LIN {X 0,Y 539.25,Z 1008.036,A -85,B 0,C 180,E1 3968.069,E2 3968.069} C_VEL
LIN {X 0,Y 539.667,Z 991.588,A -85,B 0,C 180,E1 3971.094,E2 3971.094} C_VEL
LIN {X 0,Y 540.295,Z 970.206,A -85,B 0,C 180,E1 3973.778,E2 3973.778} C_VEL
LIN {X 0,Y 541.178,Z 945.142,A -85,B 0,C 180,E1 3975.97,E2 3975.97} C_VEL
LIN {X 0,Y 542.037,Z 916.074,A -85,B 0,C 180,E1 3977.682,E2 3977.682} C_VEL
LIN {X 0,Y 542.64,Z 884.653,A -85,B 0,C 180,E1 3978.783,E2 3978.783} C_VEL
LIN {X 0,Y 541.923,Z 855.869,A -85,B 0,C 180,E1 3979.307,E2 3979.307} C_VEL
LIN {X 0,Y 538.385,Z 843.44,A -85,B 0,C 180,E1 3979.641,E2 3979.641} C_VEL
LIN {X 0,Y 538.323,Z 843.44,A -85,B 0,C 180,E1 3984.951,E2 3984.951} C_VEL
LIN {X 0,Y 538.286,Z 843.44,A -85,B 0,C 180,E1 3990.414,E2 3990.414} C_VEL
LIN {X 0,Y 538.342,Z 843.44,A -85,B 0,C 180,E1 3996.196,E2 3996.196} C_VEL
LIN {X 0,Y 538.103,Z 843.44,A -85,B 0,C 180,E1 4002.471,E2 4002.471} C_VEL
LIN {X 0,Y 538.121,Z 843.44,A -85,B 0,C 180,E1 4007.522,E2 4007.522} C_VEL
LIN {X 0,Y 538.444,Z 843.44,A -85,B 0,C 180,E1 4013.804,E2 4013.804} C_VEL
LIN {X 0,Y 538.555,Z 844.13,A -85,B 0,C 180,E1 4016.198,E2 4016.198} C_VEL
LIN {X 0,Y 549.167,Z 867.562,A -85,B 0,C 180,E1 4017.292,E2 4017.292} C_VEL
LIN {X 0,Y 548.845,Z 915.281,A -85,B 0,C 180,E1 4018.203,E2 4018.203} C_VEL
LIN {X 0,Y 547.509,Z 954.361,A -85,B 0,C 180,E1 4019.575,E2 4019.575} C_VEL
LIN {X 0,Y 545.893,Z 988.921,A -85,B 0,C 180,E1 4021.38,E2 4021.38} C_VEL
LIN {X 0,Y 543.954,Z 1023.542,A -85,B 0,C 180,E1 4023.86,E2 4023.86} C_VEL
LIN {X 0,Y 542.252,Z 1054.192,A -85,B 0,C 180,E1 4026.77,E2 4026.77} C_VEL
LIN {X 0,Y 540.773,Z 1081.673,A -85,B 0,C 180,E1 4030.169,E2 4030.169} C_VEL
LIN {X 0,Y 539.773,Z 1104.705,A -85,B 0,C 180,E1 4033.918,E2 4033.918} C_VEL
LIN {X 0,Y 539.188,Z 1122.492,A -85,B 0,C 180,E1 4037.841,E2 4037.841} C_VEL
LIN {X 0,Y 539.047,Z 1134.255,A -85,B 0,C 180,E1 4041.519,E2 4041.519} C_VEL
LIN {X 0,Y 538.908,Z 1141.5,A -85,B 0,C 180,E1 4045.164,E2 4045.164} C_VEL
LIN {X 0,Y 538.866,Z 1144.612,A -85,B 0,C 180,E1 4048.389,E2 4048.389} C_VEL
LIN {X 0,Y 538.972,Z 1144.555,A -85,B 0,C 180,E1 4051.609,E2 4051.609} C_VEL
LIN {X 0,Y 538.984,Z 1140.149,A -85,B 0,C 180,E1 4055.642,E2 4055.642} C_VEL
LIN {X 0,Y 539.118,Z 1130.585,A -85,B 0,C 180,E1 4059.701,E2 4059.701} C_VEL
LIN {X 0,Y 539.5,Z 1115.458,A -85,B 0,C 180,E1 4063.786,E2 4063.786} C_VEL
LIN {X 0,Y 540.206,Z 1095.274,A -85,B 0,C 180,E1 4067.665,E2 4067.665} C_VEL
LIN {X 0,Y 541.512,Z 1068.316,A -85,B 0,C 180,E1 4071.506,E2 4071.506} C_VEL
LIN {X 0,Y 543.119,Z 1038.564,A -85,B 0,C 180,E1 4074.719,E2 4074.719} C_VEL
LIN {X 0,Y 545.035,Z 1004.579,A -85,B 0,C 180,E1 4077.497,E2 4077.497} C_VEL
LIN {X 0,Y 546.848,Z 969.441,A -85,B 0,C 180,E1 4079.619,E2 4079.619} C_VEL
LIN {X 0,Y 548.311,Z 933.853,A -85,B 0,C 180,E1 4081.138,E2 4081.138} C_VEL
LIN {X 0,Y 549.352,Z 895.087,A -85,B 0,C 180,E1 4082.16,E2 4082.16} C_VEL
LIN {X 0,Y 548.858,Z 867.054,A -85,B 0,C 180,E1 4082.647,E2 4082.647} C_VEL
LIN {X 0,Y 538.256,Z 843.44,A -85,B 0,C 180,E1 4083.79,E2 4083.79} C_VEL
LIN {X 0,Y 538.332,Z 843.44,A -85,B 0,C 180,E1 4088.226,E2 4088.226} C_VEL
LIN {X 0,Y 538.212,Z 843.44,A -85,B 0,C 180,E1 4094.693,E2 4094.693} C_VEL
LIN {X 0,Y 538.217,Z 843.44,A -85,B 0,C 180,E1 4099.688,E2 4099.688} C_VEL
LIN {X 0,Y 538.184,Z 843.44,A -85,B 0,C 180,E1 4105.764,E2 4105.764} C_VEL
LIN {X 0,Y 538.293,Z 843.44,A -85,B 0,C 180,E1 4111.438,E2 4111.438} C_VEL
LIN {X 0,Y 538.435,Z 843.44,A -85,B 0,C 180,E1 4116.819,E2 4116.819} C_VEL
LIN {X 0,Y 538.559,Z 843.44,A -85,B 0,C 180,E1 4121.989,E2 4121.989} C_VEL
LIN {X 0,Y 538.664,Z 843.44,A -85,B 0,C 180,E1 4127.007,E2 4127.007} C_VEL
LIN {X 0,Y 538.668,Z 843.44,A -85,B 0,C 180,E1 4131.922,E2 4131.922} C_VEL
LIN {X 0,Y 538.803,Z 843.44,A -85,B 0,C 180,E1 4136.779,E2 4136.779} C_VEL
LIN {X 0,Y 538.914,Z 843.44,A -85,B 0,C 180,E1 4141.611,E2 4141.611} C_VEL
LIN {X 0,Y 538.794,Z 843.44,A -85,B 0,C 180,E1 4146.454,E2 4146.454} C_VEL
LIN {X 0,Y 538.518,Z 843.44,A -85,B 0,C 180,E1 4152.998,E2 4152.998} C_VEL
LIN {X 0,Y 538.458,Z 843.44,A -85,B 0,C 180,E1 4158.017,E2 4158.017} C_VEL
LIN {X 0,Y 538.431,Z 843.44,A -85,B 0,C 180,E1 4163.182,E2 4163.182} C_VEL
LIN {X 0,Y 538.42,Z 843.44,A -85,B 0,C 180,E1 4165.122,E2 4165.122} C_VEL
LIN {X 0,Y 537.116,Z 843.44,A -85,B 0,C 180,E1 4166.044,E2 4166.044} C_VEL
LIN {X 0,Y 530.442,Z 843.44,A -85,B 0,C 180,E1 4168.554,E2 4168.554} C_VEL
LIN {X 0,Y 530.36,Z 843.44,A -85,B 0,C 180,E1 4168.792,E2 4168.792} C_VEL
LIN {X 0,Y 530.3,Z 843.44,A -85,B 0,C 180,E1 4174.819,E2 4174.819} C_VEL
LIN {X 0,Y 530.294,Z 843.44,A -85,B 0,C 180,E1 4181.044,E2 4181.044} C_VEL
LIN {X 0,Y 530.296,Z 843.44,A -85,B 0,C 180,E1 4186.745,E2 4186.745} C_VEL
LIN {X 0,Y 530.38,Z 844.061,A -85,B 0,C 180,E1 4190.548,E2 4190.548} C_VEL
LIN {X 0,Y 546.247,Z 875.945,A -85,B 0,C 180,E1 4192.425,E2 4192.425} C_VEL
LIN {X 0,Y 545.089,Z 919.849,A -85,B 0,C 180,E1 4193.364,E2 4193.364} C_VEL
LIN {X 0,Y 543.337,Z 959.293,A -85,B 0,C 180,E1 4194.829,E2 4194.829} C_VEL
LIN {X 0,Y 541.124,Z 997.278,A -85,B 0,C 180,E1 4196.867,E2 4196.867} C_VEL
LIN {X 0,Y 538.391,Z 1035.857,A -85,B 0,C 180,E1 4199.684,E2 4199.684} C_VEL
LIN {X 0,Y 535.813,Z 1071.337,A -85,B 0,C 180,E1 4203.12,E2 4203.12} C_VEL
LIN {X 0,Y 533.767,Z 1102.204,A -85,B 0,C 180,E1 4207.015,E2 4207.015} C_VEL
LIN {X 0,Y 532.286,Z 1127.302,A -85,B 0,C 180,E1 4211.122,E2 4211.122} C_VEL
LIN {X 0,Y 531.574,Z 1145.987,A -85,B 0,C 180,E1 4215.147,E2 4215.147} C_VEL
LIN {X 0,Y 531.16,Z 1160,A -85,B 0,C 180,E1 4219.272,E2 4219.272} C_VEL
LIN {X 0,Y 531.066,Z 1169.479,A -85,B 0,C 180,E1 4223.452,E2 4223.452} C_VEL
LIN {X 0,Y 530.978,Z 1173.628,A -85,B 0,C 180,E1 4226.731,E2 4226.731} C_VEL
LIN {X 0,Y 530.953,Z 1175,A -85,B 0,C 180,E1 4230.001,E2 4230.001} C_VEL
LIN {X 0,Y 530.956,Z 1173.247,A -85,B 0,C 180,E1 4233.638,E2 4233.638} C_VEL
LIN {X 0,Y 531.102,Z 1166.328,A -85,B 0,C 180,E1 4238.196,E2 4238.196} C_VEL
LIN {X 0,Y 531.263,Z 1155.088,A -85,B 0,C 180,E1 4242.343,E2 4242.343} C_VEL
LIN {X 0,Y 531.834,Z 1138.762,A -85,B 0,C 180,E1 4246.542,E2 4246.542} C_VEL
LIN {X 0,Y 532.945,Z 1116.87,A -85,B 0,C 180,E1 4250.718,E2 4250.718} C_VEL
LIN {X 0,Y 534.62,Z 1089.193,A -85,B 0,C 180,E1 4254.753,E2 4254.753} C_VEL
LIN {X 0,Y 536.83,Z 1057.678,A -85,B 0,C 180,E1 4258.313,E2 4258.313} C_VEL
LIN {X 0,Y 539.421,Z 1021.619,A -85,B 0,C 180,E1 4261.454,E2 4261.454} C_VEL
LIN {X 0,Y 542.046,Z 982.156,A -85,B 0,C 180,E1 4264.028,E2 4264.028} C_VEL
LIN {X 0,Y 544.325,Z 941.057,A -85,B 0,C 180,E1 4265.927,E2 4265.927} C_VEL
LIN {X 0,Y 545.815,Z 903.152,A -85,B 0,C 180,E1 4267.057,E2 4267.057} C_VEL
LIN {X 0,Y 545.931,Z 873.898,A -85,B 0,C 180,E1 4267.634,E2 4267.634} C_VEL
LIN {X 0,Y 530.636,Z 845.115,A -85,B 0,C 180,E1 4269.411,E2 4269.411} C_VEL
LIN {X 0,Y 530.457,Z 843.44,A -85,B 0,C 180,E1 4269.456,E2 4269.456} C_VEL
LIN {X 0,Y 530.126,Z 843.44,A -85,B 0,C 180,E1 4275.566,E2 4275.566} C_VEL
LIN {X 0,Y 530.325,Z 843.44,A -85,B 0,C 180,E1 4281.093,E2 4281.093} C_VEL
LIN {X 0,Y 530.43,Z 843.44,A -85,B 0,C 180,E1 4287.159,E2 4287.159} C_VEL
LIN {X 0,Y 530.426,Z 843.44,A -85,B 0,C 180,E1 4292.827,E2 4292.827} C_VEL
LIN {X 0,Y 530.381,Z 843.44,A -85,B 0,C 180,E1 4298.217,E2 4298.217} C_VEL
LIN {X 0,Y 530.241,Z 843.44,A -85,B 0,C 180,E1 4299.962,E2 4299.962} C_VEL
LIN {X 0,Y 535.362,Z 865.662,A -85,B 0,C 180,E1 4300.493,E2 4300.493} C_VEL
LIN {X 0,Y 534.887,Z 898.665,A -85,B 0,C 180,E1 4301.266,E2 4301.266} C_VEL
LIN {X 0,Y 534.068,Z 927.663,A -85,B 0,C 180,E1 4302.577,E2 4302.577} C_VEL
LIN {X 0,Y 533.058,Z 956.085,A -85,B 0,C 180,E1 4304.579,E2 4304.579} C_VEL
LIN {X 0,Y 532.241,Z 978.331,A -85,B 0,C 180,E1 4306.846,E2 4306.846} C_VEL
LIN {X 0,Y 531.653,Z 997.827,A -85,B 0,C 180,E1 4309.667,E2 4309.667} C_VEL
LIN {X 0,Y 531.371,Z 1011.704,A -85,B 0,C 180,E1 4312.633,E2 4312.633} C_VEL
LIN {X 0,Y 531.191,Z 1020.396,A -85,B 0,C 180,E1 4315.596,E2 4315.596} C_VEL
LIN {X 0,Y 531.1,Z 1024.385,A -85,B 0,C 180,E1 4318.366,E2 4318.366} C_VEL
LIN {X 0,Y 531.096,Z 1024.309,A -85,B 0,C 180,E1 4321.633,E2 4321.633} C_VEL
LIN {X 0,Y 531.2,Z 1019.034,A -85,B 0,C 180,E1 4324.904,E2 4324.904} C_VEL
LIN {X 0,Y 531.382,Z 1008.039,A -85,B 0,C 180,E1 4328.189,E2 4328.189} C_VEL
LIN {X 0,Y 531.844,Z 991.591,A -85,B 0,C 180,E1 4331.26,E2 4331.26} C_VEL
LIN {X 0,Y 532.563,Z 970.21,A -85,B 0,C 180,E1 4333.982,E2 4333.982} C_VEL
LIN {X 0,Y 533.528,Z 944.229,A -85,B 0,C 180,E1 4336.272,E2 4336.272} C_VEL
LIN {X 0,Y 534.512,Z 914.964,A -85,B 0,C 180,E1 4337.993,E2 4337.993} C_VEL
LIN {X 0,Y 535.152,Z 885.089,A -85,B 0,C 180,E1 4339.045,E2 4339.045} C_VEL
LIN {X 0,Y 534.775,Z 858.414,A -85,B 0,C 180,E1 4339.54,E2 4339.54} C_VEL
LIN {X 0,Y 530.44,Z 843.44,A -85,B 0,C 180,E1 4339.92,E2 4339.92} C_VEL
LIN {X 0,Y 530.42,Z 843.44,A -85,B 0,C 180,E1 4345.348,E2 4345.348} C_VEL
LIN {X 0,Y 530.335,Z 843.44,A -85,B 0,C 180,E1 4351.071,E2 4351.071} C_VEL
LIN {X 0,Y 530.359,Z 843.44,A -85,B 0,C 180,E1 4356.928,E2 4356.928} C_VEL
LIN {X 0,Y 530.126,Z 843.44,A -85,B 0,C 180,E1 4363.266,E2 4363.266} C_VEL
LIN {X 0,Y 530.268,Z 843.44,A -85,B 0,C 180,E1 4368.947,E2 4368.947} C_VEL
LIN {X 0,Y 530.543,Z 843.44,A -85,B 0,C 180,E1 4375.427,E2 4375.427} C_VEL
LIN {X 0,Y 530.554,Z 843.44,A -85,B 0,C 180,E1 4375.604,E2 4375.604} C_VEL
LIN {X 0,Y 542.545,Z 871.557,A -85,B 0,C 180,E1 4376.904,E2 4376.904} C_VEL
LIN {X 0,Y 542.059,Z 916.69,A -85,B 0,C 180,E1 4377.801,E2 4377.801} C_VEL
LIN {X 0,Y 540.643,Z 954.411,A -85,B 0,C 180,E1 4379.15,E2 4379.15} C_VEL
LIN {X 0,Y 538.857,Z 988.917,A -85,B 0,C 180,E1 4380.972,E2 4380.972} C_VEL
LIN {X 0,Y 536.689,Z 1023.761,A -85,B 0,C 180,E1 4383.499,E2 4383.499} C_VEL
LIN {X 0,Y 534.806,Z 1054.184,A -85,B 0,C 180,E1 4386.427,E2 4386.427} C_VEL
LIN {X 0,Y 533.143,Z 1081.644,A -85,B 0,C 180,E1 4389.869,E2 4389.869} C_VEL
LIN {X 0,Y 532.025,Z 1104.702,A -85,B 0,C 180,E1 4393.677,E2 4393.677} C_VEL
LIN {X 0,Y 531.351,Z 1122.49,A -85,B 0,C 180,E1 4397.659,E2 4397.659} C_VEL
LIN {X 0,Y 531.161,Z 1134.254,A -85,B 0,C 180,E1 4401.392,E2 4401.392} C_VEL
LIN {X 0,Y 531.02,Z 1141.499,A -85,B 0,C 180,E1 4405.092,E2 4405.092} C_VEL
LIN {X 0,Y 530.964,Z 1144.612,A -85,B 0,C 180,E1 4408.365,E2 4408.365} C_VEL
LIN {X 0,Y 531.067,Z 1144.555,A -85,B 0,C 180,E1 4411.633,E2 4411.633} C_VEL
LIN {X 0,Y 531.079,Z 1140.151,A -85,B 0,C 180,E1 4415.726,E2 4415.726} C_VEL
LIN {X 0,Y 531.244,Z 1130.587,A -85,B 0,C 180,E1 4419.846,E2 4419.846} C_VEL
LIN {X 0,Y 531.659,Z 1114.651,A -85,B 0,C 180,E1 4424.182,E2 4424.182} C_VEL
LIN {X 0,Y 532.574,Z 1093.495,A -85,B 0,C 180,E1 4428.223,E2 4428.223} C_VEL
LIN {X 0,Y 533.995,Z 1067.089,A -85,B 0,C 180,E1 4431.978,E2 4431.978} C_VEL
LIN {X 0,Y 535.838,Z 1036.864,A -85,B 0,C 180,E1 4435.244,E2 4435.244} C_VEL
LIN {X 0,Y 537.938,Z 1003.455,A -85,B 0,C 180,E1 4437.976,E2 4437.976} C_VEL
LIN {X 0,Y 539.961,Z 967.997,A -85,B 0,C 180,E1 4440.115,E2 4440.115} C_VEL
LIN {X 0,Y 541.596,Z 932.081,A -85,B 0,C 180,E1 4441.632,E2 4441.632} C_VEL
LIN {X 0,Y 542.685,Z 895.255,A -85,B 0,C 180,E1 4442.601,E2 4442.601} C_VEL
LIN {X 0,Y 542.233,Z 869.608,A -85,B 0,C 180,E1 4443.058,E2 4443.058} C_VEL
LIN {X 0,Y 530.33,Z 843.44,A -85,B 0,C 180,E1 4444.378,E2 4444.378} C_VEL
LIN {X 0,Y 530.31,Z 843.44,A -85,B 0,C 180,E1 4449.575,E2 4449.575} C_VEL
LIN {X 0,Y 530.304,Z 843.44,A -85,B 0,C 180,E1 4455.544,E2 4455.544} C_VEL
LIN {X 0,Y 530.257,Z 843.44,A -85,B 0,C 180,E1 4461.089,E2 4461.089} C_VEL
LIN {X 0,Y 530.268,Z 843.44,A -85,B 0,C 180,E1 4467.15,E2 4467.15} C_VEL
LIN {X 0,Y 530.43,Z 843.44,A -85,B 0,C 180,E1 4472.829,E2 4472.829} C_VEL
LIN {X 0,Y 530.578,Z 843.44,A -85,B 0,C 180,E1 4478.227,E2 4478.227} C_VEL
LIN {X 0,Y 530.67,Z 843.44,A -85,B 0,C 180,E1 4483.425,E2 4483.425} C_VEL
LIN {X 0,Y 530.676,Z 843.44,A -85,B 0,C 180,E1 4488.481,E2 4488.481} C_VEL
LIN {X 0,Y 530.714,Z 843.44,A -85,B 0,C 180,E1 4493.449,E2 4493.449} C_VEL
LIN {X 0,Y 530.763,Z 843.44,A -85,B 0,C 180,E1 4498.366,E2 4498.366} C_VEL
LIN {X 0,Y 530.765,Z 843.44,A -85,B 0,C 180,E1 4503.271,E2 4503.271} C_VEL
LIN {X 0,Y 530.657,Z 843.44,A -85,B 0,C 180,E1 4508.202,E2 4508.202} C_VEL
LIN {X 0,Y 530.555,Z 843.44,A -85,B 0,C 180,E1 4513.999,E2 4513.999} C_VEL
LIN {X 0,Y 530.537,Z 843.44,A -85,B 0,C 180,E1 4520.026,E2 4520.026} C_VEL
LIN {X 0,Y 530.536,Z 843.44,A -85,B 0,C 180,E1 4525.344,E2 4525.344} C_VEL
LIN {X 0,Y 530.36,Z 843.44,A -85,B 0,C 180,E1 4528.792,E2 4528.792} C_VEL
LIN {X 0,Y 527.819,Z 843.44,A -85,B 0,C 180,E1 4530.18,E2 4530.18} C_VEL
LIN {X 0,Y 522.427,Z 843.44,A -85,B 0,C 180,E1 4532.26,E2 4532.26} C_VEL
LIN {X 0,Y 522.35,Z 843.44,A -85,B 0,C 180,E1 4532.501,E2 4532.501} C_VEL
LIN {X 0,Y 522.357,Z 843.44,A -85,B 0,C 180,E1 4538.499,E2 4538.499} C_VEL
LIN {X 0,Y 522.418,Z 843.44,A -85,B 0,C 180,E1 4544.069,E2 4544.069} C_VEL
LIN {X 0,Y 522.382,Z 844.116,A -85,B 0,C 180,E1 4549.825,E2 4549.825} C_VEL
LIN {X 0,Y 539.951,Z 879.393,A -85,B 0,C 180,E1 4551.966,E2 4551.966} C_VEL
LIN {X 0,Y 538.635,Z 922.756,A -85,B 0,C 180,E1 4552.945,E2 4552.945} C_VEL
LIN {X 0,Y 536.659,Z 962.005,A -85,B 0,C 180,E1 4554.464,E2 4554.464} C_VEL
LIN {X 0,Y 534.198,Z 999.236,A -85,B 0,C 180,E1 4556.521,E2 4556.521} C_VEL
LIN {X 0,Y 531.304,Z 1036.601,A -85,B 0,C 180,E1 4559.306,E2 4559.306} C_VEL
LIN {X 0,Y 528.494,Z 1071.337,A -85,B 0,C 180,E1 4562.717,E2 4562.717} C_VEL
LIN {X 0,Y 526.312,Z 1101.078,A -85,B 0,C 180,E1 4566.498,E2 4566.498} C_VEL
LIN {X 0,Y 524.669,Z 1126.193,A -85,B 0,C 180,E1 4570.618,E2 4570.618} C_VEL
LIN {X 0,Y 523.746,Z 1145.985,A -85,B 0,C 180,E1 4574.92,E2 4574.92} C_VEL
LIN {X 0,Y 523.289,Z 1159.852,A -85,B 0,C 180,E1 4579.055,E2 4579.055} C_VEL
LIN {X 0,Y 523.163,Z 1169.479,A -85,B 0,C 180,E1 4583.353,E2 4583.353} C_VEL
LIN {X 0,Y 523.098,Z 1173.628,A -85,B 0,C 180,E1 4586.682,E2 4586.682} C_VEL
LIN {X 0,Y 523.065,Z 1175,A -85,B 0,C 180,E1 4590.001,E2 4590.001} C_VEL
LIN {X 0,Y 523.097,Z 1173.627,A -85,B 0,C 180,E1 4593.32,E2 4593.32} C_VEL
LIN {X 0,Y 523.255,Z 1167.915,A -85,B 0,C 180,E1 4597.483,E2 4597.483} C_VEL
LIN {X 0,Y 523.353,Z 1157.769,A -85,B 0,C 180,E1 4601.685,E2 4601.685} C_VEL
LIN {X 0,Y 523.901,Z 1142.484,A -85,B 0,C 180,E1 4605.937,E2 4605.937} C_VEL
LIN {X 0,Y 524.966,Z 1121.368,A -85,B 0,C 180,E1 4610.25,E2 4610.25} C_VEL
LIN {X 0,Y 526.718,Z 1095.264,A -85,B 0,C 180,E1 4614.311,E2 4614.311} C_VEL
LIN {X 0,Y 529.005,Z 1065.179,A -85,B 0,C 180,E1 4617.949,E2 4617.949} C_VEL
LIN {X 0,Y 531.717,Z 1031.06,A -85,B 0,C 180,E1 4621.158,E2 4621.158} C_VEL
LIN {X 0,Y 534.514,Z 993.918,A -85,B 0,C 180,E1 4623.82,E2 4623.82} C_VEL
LIN {X 0,Y 537.167,Z 954.369,A -85,B 0,C 180,E1 4625.886,E2 4625.886} C_VEL
LIN {X 0,Y 539.088,Z 913.257,A -85,B 0,C 180,E1 4627.323,E2 4627.323} C_VEL
LIN {X 0,Y 539.566,Z 876.644,A -85,B 0,C 180,E1 4628.111,E2 4628.111} C_VEL
LIN {X 0,Y 522.625,Z 844.942,A -85,B 0,C 180,E1 4630.139,E2 4630.139} C_VEL
LIN {X 0,Y 522.433,Z 843.44,A -85,B 0,C 180,E1 4630.286,E2 4630.286} C_VEL
LIN {X 0,Y 522.248,Z 843.44,A -85,B 0,C 180,E1 4636.455,E2 4636.455} C_VEL
LIN {X 0,Y 522.424,Z 843.44,A -85,B 0,C 180,E1 4642.513,E2 4642.513} C_VEL
LIN {X 0,Y 522.484,Z 843.44,A -85,B 0,C 180,E1 4648.562,E2 4648.562} C_VEL
LIN {X 0,Y 522.48,Z 843.44,A -85,B 0,C 180,E1 4654.237,E2 4654.237} C_VEL
LIN {X 0,Y 522.342,Z 843.44,A -85,B 0,C 180,E1 4659.689,E2 4659.689} C_VEL
LIN {X 0,Y 527.927,Z 865.615,A -85,B 0,C 180,E1 4660.207,E2 4660.207} C_VEL
LIN {X 0,Y 527.386,Z 898.235,A -85,B 0,C 180,E1 4660.976,E2 4660.976} C_VEL
LIN {X 0,Y 526.488,Z 927.634,A -85,B 0,C 180,E1 4662.317,E2 4662.317} C_VEL
LIN {X 0,Y 525.393,Z 955.804,A -85,B 0,C 180,E1 4664.326,E2 4664.326} C_VEL
LIN {X 0,Y 524.471,Z 978.32,A -85,B 0,C 180,E1 4666.647,E2 4666.647} C_VEL
LIN {X 0,Y 523.838,Z 997.943,A -85,B 0,C 180,E1 4669.532,E2 4669.532} C_VEL
LIN {X 0,Y 523.494,Z 1011.693,A -85,B 0,C 180,E1 4672.522,E2 4672.522} C_VEL
LIN {X 0,Y 523.3,Z 1020.394,A -85,B 0,C 180,E1 4675.53,E2 4675.53} C_VEL
LIN {X 0,Y 523.215,Z 1024.383,A -85,B 0,C 180,E1 4678.341,E2 4678.341} C_VEL
LIN {X 0,Y 523.212,Z 1024.308,A -85,B 0,C 180,E1 4681.657,E2 4681.657} C_VEL
LIN {X 0,Y 523.303,Z 1019.036,A -85,B 0,C 180,E1 4684.978,E2 4684.978} C_VEL
LIN {X 0,Y 523.52,Z 1008.042,A -85,B 0,C 180,E1 4688.313,E2 4688.313} C_VEL
LIN {X 0,Y 524.013,Z 992.184,A -85,B 0,C 180,E1 4691.339,E2 4691.339} C_VEL
LIN {X 0,Y 524.771,Z 972.163,A -85,B 0,C 180,E1 4693.98,E2 4693.98} C_VEL
LIN {X 0,Y 525.8,Z 947.035,A -85,B 0,C 180,E1 4696.303,E2 4696.303} C_VEL
LIN {X 0,Y 526.87,Z 918.222,A -85,B 0,C 180,E1 4698.1,E2 4698.1} C_VEL
LIN {X 0,Y 527.659,Z 888.347,A -85,B 0,C 180,E1 4699.245,E2 4699.245} C_VEL
LIN {X 0,Y 527.209,Z 859.544,A -85,B 0,C 180,E1 4699.817,E2 4699.817} C_VEL
LIN {X 0,Y 522.524,Z 843.44,A -85,B 0,C 180,E1 4700.262,E2 4700.262} C_VEL
LIN {X 0,Y 522.424,Z 843.44,A -85,B 0,C 180,E1 4706.041,E2 4706.041} C_VEL
LIN {X 0,Y 522.414,Z 843.44,A -85,B 0,C 180,E1 4711.441,E2 4711.441} C_VEL
LIN {X 0,Y 522.393,Z 843.44,A -85,B 0,C 180,E1 4717.487,E2 4717.487} C_VEL
LIN {X 0,Y 522.219,Z 843.44,A -85,B 0,C 180,E1 4723.542,E2 4723.542} C_VEL
LIN {X 0,Y 522.372,Z 843.44,A -85,B 0,C 180,E1 4728.896,E2 4728.896} C_VEL
LIN {X 0,Y 522.596,Z 843.44,A -85,B 0,C 180,E1 4734.992,E2 4734.992} C_VEL
LIN {X 0,Y 535.918,Z 873.698,A -85,B 0,C 180,E1 4736.476,E2 4736.476} C_VEL
LIN {X 0,Y 535.322,Z 917.865,A -85,B 0,C 180,E1 4737.382,E2 4737.382} C_VEL
LIN {X 0,Y 533.685,Z 956.285,A -85,B 0,C 180,E1 4738.795,E2 4738.795} C_VEL
LIN {X 0,Y 531.594,Z 992.09,A -85,B 0,C 180,E1 4740.755,E2 4740.755} C_VEL
LIN {X 0,Y 529.23,Z 1026.349,A -85,B 0,C 180,E1 4743.331,E2 4743.331} C_VEL
LIN {X 0,Y 527.099,Z 1057.721,A -85,B 0,C 180,E1 4746.475,E2 4746.475} C_VEL
LIN {X 0,Y 525.336,Z 1084.483,A -85,B 0,C 180,E1 4749.984,E2 4749.984} C_VEL
LIN {X 0,Y 524.121,Z 1106.876,A -85,B 0,C 180,E1 4753.855,E2 4753.855} C_VEL
LIN {X 0,Y 523.455,Z 1124.026,A -85,B 0,C 180,E1 4757.894,E2 4757.894} C_VEL
LIN {X 0,Y 523.244,Z 1135.215,A -85,B 0,C 180,E1 4761.68,E2 4761.68} C_VEL
LIN {X 0,Y 523.12,Z 1141.499,A -85,B 0,C 180,E1 4765.018,E2 4765.018} C_VEL
LIN {X 0,Y 523.06,Z 1144.611,A -85,B 0,C 180,E1 4768.34,E2 4768.34} C_VEL
LIN {X 0,Y 523.178,Z 1144.556,A -85,B 0,C 180,E1 4771.658,E2 4771.658} C_VEL
LIN {X 0,Y 523.189,Z 1140.152,A -85,B 0,C 180,E1 4775.813,E2 4775.813} C_VEL
LIN {X 0,Y 523.361,Z 1130.589,A -85,B 0,C 180,E1 4779.996,E2 4779.996} C_VEL
LIN {X 0,Y 523.817,Z 1115.133,A -85,B 0,C 180,E1 4784.288,E2 4784.288} C_VEL
LIN {X 0,Y 524.904,Z 1093.498,A -85,B 0,C 180,E1 4788.499,E2 4788.499} C_VEL
LIN {X 0,Y 526.412,Z 1067.473,A -85,B 0,C 180,E1 4792.264,E2 4792.264} C_VEL
LIN {X 0,Y 528.489,Z 1037.362,A -85,B 0,C 180,E1 4795.572,E2 4795.572} C_VEL
LIN {X 0,Y 530.772,Z 1004.033,A -85,B 0,C 180,E1 4798.344,E2 4798.344} C_VEL
LIN {X 0,Y 533.009,Z 968.113,A -85,B 0,C 180,E1 4800.543,E2 4800.543} C_VEL
LIN {X 0,Y 534.859,Z 931.791,A -85,B 0,C 180,E1 4802.089,E2 4802.089} C_VEL
LIN {X 0,Y 536.022,Z 894.735,A -85,B 0,C 180,E1 4803.068,E2 4803.068} C_VEL
LIN {X 0,Y 535.537,Z 872.12,A -85,B 0,C 180,E1 4803.486,E2 4803.486} C_VEL
LIN {X 0,Y 522.398,Z 843.44,A -85,B 0,C 180,E1 4805.018,E2 4805.018} C_VEL
LIN {X 0,Y 522.397,Z 843.44,A -85,B 0,C 180,E1 4811.107,E2 4811.107} C_VEL
LIN {X 0,Y 522.433,Z 843.44,A -85,B 0,C 180,E1 4816.431,E2 4816.431} C_VEL
LIN {X 0,Y 522.312,Z 843.44,A -85,B 0,C 180,E1 4822.506,E2 4822.506} C_VEL
LIN {X 0,Y 522.358,Z 843.44,A -85,B 0,C 180,E1 4828.555,E2 4828.555} C_VEL
LIN {X 0,Y 522.561,Z 843.44,A -85,B 0,C 180,E1 4834.243,E2 4834.243} C_VEL
LIN {X 0,Y 522.689,Z 843.44,A -85,B 0,C 180,E1 4839.662,E2 4839.662} C_VEL
LIN {X 0,Y 522.798,Z 843.44,A -85,B 0,C 180,E1 4844.894,E2 4844.894} C_VEL
LIN {X 0,Y 522.809,Z 843.44,A -85,B 0,C 180,E1 4851.219,E2 4851.219} C_VEL
LIN {X 0,Y 523.027,Z 843.44,A -85,B 0,C 180,E1 4856.682,E2 4856.682} C_VEL
LIN {X 0,Y 523.095,Z 843.44,A -85,B 0,C 180,E1 4861.659,E2 4861.659} C_VEL
LIN {X 0,Y 522.953,Z 843.44,A -85,B 0,C 180,E1 4866.651,E2 4866.651} C_VEL
LIN {X 0,Y 522.759,Z 843.44,A -85,B 0,C 180,E1 4871.697,E2 4871.697} C_VEL
LIN {X 0,Y 522.618,Z 843.44,A -85,B 0,C 180,E1 4877.047,E2 4877.047} C_VEL
LIN {X 0,Y 522.615,Z 843.44,A -85,B 0,C 180,E1 4882.124,E2 4882.124} C_VEL
LIN {X 0,Y 522.499,Z 843.44,A -85,B 0,C 180,E1 4887.621,E2 4887.621} C_VEL
LIN {X 0,Y 522.35,Z 843.44,A -85,B 0,C 180,E1 4892.501,E2 4892.501} C_VEL
LIN {X 0,Y 519.889,Z 843.44,A -85,B 0,C 180,E1 4893.915,E2 4893.915} C_VEL
LIN {X 0,Y 514.52,Z 843.44,A -85,B 0,C 180,E1 4896.034,E2 4896.034} C_VEL
LIN {X 0,Y 514.418,Z 843.44,A -85,B 0,C 180,E1 4896.279,E2 4896.279} C_VEL
LIN {X 0,Y 514.476,Z 843.44,A -85,B 0,C 180,E1 4902.629,E2 4902.629} C_VEL
LIN {X 0,Y 514.457,Z 843.978,A -85,B 0,C 180,E1 4909.177,E2 4909.177} C_VEL
LIN {X 0,Y 527.261,Z 868.244,A -85,B 0,C 180,E1 4910.687,E2 4910.687} C_VEL
LIN {X 0,Y 533.59,Z 880.607,A -85,B 0,C 180,E1 4911.45,E2 4911.45} C_VEL
LIN {X 0,Y 532.173,Z 925.769,A -85,B 0,C 180,E1 4912.518,E2 4912.518} C_VEL
LIN {X 0,Y 529.638,Z 969.015,A -85,B 0,C 180,E1 4914.288,E2 4914.288} C_VEL
LIN {X 0,Y 526.509,Z 1010.216,A -85,B 0,C 180,E1 4916.771,E2 4916.771} C_VEL
LIN {X 0,Y 523.22,Z 1048.534,A -85,B 0,C 180,E1 4919.933,E2 4919.933} C_VEL
LIN {X 0,Y 520.413,Z 1081.104,A -85,B 0,C 180,E1 4923.456,E2 4923.456} C_VEL
LIN {X 0,Y 518.058,Z 1111.031,A -85,B 0,C 180,E1 4927.67,E2 4927.67} C_VEL
LIN {X 0,Y 516.557,Z 1134.744,A -85,B 0,C 180,E1 4932.054,E2 4932.054} C_VEL
LIN {X 0,Y 515.734,Z 1153.745,A -85,B 0,C 180,E1 4936.849,E2 4936.849} C_VEL
LIN {X 0,Y 515.351,Z 1166.332,A -85,B 0,C 180,E1 4941.553,E2 4941.553} C_VEL
LIN {X 0,Y 515.323,Z 1171.905,A -85,B 0,C 180,E1 4944.944,E2 4944.944} C_VEL
LIN {X 0,Y 515.28,Z 1174.657,A -85,B 0,C 180,E1 4948.317,E2 4948.317} C_VEL
LIN {X 0,Y 515.201,Z 1173.627,A -85,B 0,C 180,E1 4953.37,E2 4953.37} C_VEL
LIN {X 0,Y 515.349,Z 1167.915,A -85,B 0,C 180,E1 4957.598,E2 4957.598} C_VEL
LIN {X 0,Y 515.484,Z 1157.769,A -85,B 0,C 180,E1 4961.866,E2 4961.866} C_VEL
LIN {X 0,Y 516.11,Z 1142.485,A -85,B 0,C 180,E1 4966.184,E2 4966.184} C_VEL
LIN {X 0,Y 517.304,Z 1121.37,A -85,B 0,C 180,E1 4970.564,E2 4970.564} C_VEL
LIN {X 0,Y 519.193,Z 1095.847,A -85,B 0,C 180,E1 4974.603,E2 4974.603} C_VEL
LIN {X 0,Y 521.774,Z 1065.169,A -85,B 0,C 180,E1 4978.372,E2 4978.372} C_VEL
LIN {X 0,Y 524.773,Z 1031.062,A -85,B 0,C 180,E1 4981.617,E2 4981.617} C_VEL
LIN {X 0,Y 527.82,Z 993.519,A -85,B 0,C 180,E1 4984.335,E2 4984.335} C_VEL
LIN {X 0,Y 530.754,Z 953.151,A -85,B 0,C 180,E1 4986.444,E2 4986.444} C_VEL
LIN {X 0,Y 532.814,Z 913.172,A -85,B 0,C 180,E1 4987.841,E2 4987.841} C_VEL
LIN {X 0,Y 533.296,Z 879.52,A -85,B 0,C 180,E1 4988.593,E2 4988.593} C_VEL
LIN {X 0,Y 514.647,Z 844.935,A -85,B 0,C 180,E1 4990.791,E2 4990.791} C_VEL
LIN {X 0,Y 514.479,Z 843.44,A -85,B 0,C 180,E1 4990.892,E2 4990.892} C_VEL
LIN {X 0,Y 514.34,Z 843.44,A -85,B 0,C 180,E1 4997.39,E2 4997.39} C_VEL
LIN {X 0,Y 514.531,Z 843.44,A -85,B 0,C 180,E1 5002.613,E2 5002.613} C_VEL
LIN {X 0,Y 514.594,Z 843.44,A -85,B 0,C 180,E1 5008.573,E2 5008.573} C_VEL
LIN {X 0,Y 514.566,Z 843.44,A -85,B 0,C 180,E1 5013.811,E2 5013.811} C_VEL
LIN {X 0,Y 514.441,Z 843.44,A -85,B 0,C 180,E1 5019.44,E2 5019.44} C_VEL
LIN {X 0,Y 520.414,Z 867.219,A -85,B 0,C 180,E1 5019.975,E2 5019.975} C_VEL
LIN {X 0,Y 519.877,Z 899.91,A -85,B 0,C 180,E1 5020.759,E2 5020.759} C_VEL
LIN {X 0,Y 518.925,Z 928.408,A -85,B 0,C 180,E1 5022.092,E2 5022.092} C_VEL
LIN {X 0,Y 517.687,Z 957.054,A -85,B 0,C 180,E1 5024.196,E2 5024.196} C_VEL
LIN {X 0,Y 516.656,Z 979.928,A -85,B 0,C 180,E1 5026.657,E2 5026.657} C_VEL
LIN {X 0,Y 515.975,Z 998.703,A -85,B 0,C 180,E1 5029.515,E2 5029.515} C_VEL
LIN {X 0,Y 515.56,Z 1013.2,A -85,B 0,C 180,E1 5032.83,E2 5032.83} C_VEL
LIN {X 0,Y 515.403,Z 1021.025,A -85,B 0,C 180,E1 5035.788,E2 5035.788} C_VEL
LIN {X 0,Y 515.314,Z 1024.381,A -85,B 0,C 180,E1 5038.316,E2 5038.316} C_VEL
LIN {X 0,Y 515.31,Z 1024.307,A -85,B 0,C 180,E1 5041.683,E2 5041.683} C_VEL
LIN {X 0,Y 515.407,Z 1019.039,A -85,B 0,C 180,E1 5045.055,E2 5045.055} C_VEL
LIN {X 0,Y 515.672,Z 1008.046,A -85,B 0,C 180,E1 5048.44,E2 5048.44} C_VEL
LIN {X 0,Y 516.182,Z 991.66,A -85,B 0,C 180,E1 5051.596,E2 5051.596} C_VEL
LIN {X 0,Y 517.127,Z 970.072,A -85,B 0,C 180,E1 5054.424,E2 5054.424} C_VEL
LIN {X 0,Y 518.313,Z 944.239,A -85,B 0,C 180,E1 5056.764,E2 5056.764} C_VEL
LIN {X 0,Y 519.433,Z 915.858,A -85,B 0,C 180,E1 5058.493,E2 5058.493} C_VEL
LIN {X 0,Y 520.197,Z 885.763,A -85,B 0,C 180,E1 5059.584,E2 5059.584} C_VEL
LIN {X 0,Y 519.832,Z 861.5,A -85,B 0,C 180,E1 5060.054,E2 5060.054} C_VEL
LIN {X 0,Y 514.592,Z 843.44,A -85,B 0,C 180,E1 5060.546,E2 5060.546} C_VEL
LIN {X 0,Y 514.521,Z 843.44,A -85,B 0,C 180,E1 5066.19,E2 5066.19} C_VEL
LIN {X 0,Y 514.535,Z 843.44,A -85,B 0,C 180,E1 5071.979,E2 5071.979} C_VEL
LIN {X 0,Y 514.457,Z 843.44,A -85,B 0,C 180,E1 5078.168,E2 5078.168} C_VEL
LIN {X 0,Y 514.33,Z 843.44,A -85,B 0,C 180,E1 5082.609,E2 5082.609} C_VEL
LIN {X 0,Y 514.462,Z 843.44,A -85,B 0,C 180,E1 5089.646,E2 5089.646} C_VEL
LIN {X 0,Y 514.65,Z 843.658,A -85,B 0,C 180,E1 5094.314,E2 5094.314} C_VEL
LIN {X 0,Y 529.357,Z 875.577,A -85,B 0,C 180,E1 5096.035,E2 5096.035} C_VEL
LIN {X 0,Y 528.643,Z 918.128,A -85,B 0,C 180,E1 5096.927,E2 5096.927} C_VEL
LIN {X 0,Y 526.924,Z 955.448,A -85,B 0,C 180,E1 5098.308,E2 5098.308} C_VEL
LIN {X 0,Y 524.688,Z 990.782,A -85,B 0,C 180,E1 5100.242,E2 5100.242} C_VEL
LIN {X 0,Y 522.106,Z 1025.071,A -85,B 0,C 180,E1 5102.821,E2 5102.821} C_VEL
LIN {X 0,Y 519.781,Z 1056.092,A -85,B 0,C 180,E1 5105.931,E2 5105.931} C_VEL
LIN {X 0,Y 517.807,Z 1083.017,A -85,B 0,C 180,E1 5109.457,E2 5109.457} C_VEL
LIN {X 0,Y 516.471,Z 1105.785,A -85,B 0,C 180,E1 5113.39,E2 5113.39} C_VEL
LIN {X 0,Y 515.698,Z 1122.486,A -85,B 0,C 180,E1 5117.278,E2 5117.278} C_VEL
LIN {X 0,Y 515.357,Z 1135.213,A -85,B 0,C 180,E1 5121.552,E2 5121.552} C_VEL
LIN {X 0,Y 515.24,Z 1141.498,A -85,B 0,C 180,E1 5124.941,E2 5124.941} C_VEL
LIN {X 0,Y 515.183,Z 1144.611,A -85,B 0,C 180,E1 5128.315,E2 5128.315} C_VEL
LIN {X 0,Y 515.197,Z 1144.104,A -85,B 0,C 180,E1 5132.432,E2 5132.432} C_VEL
LIN {X 0,Y 515.266,Z 1138.599,A -85,B 0,C 180,E1 5136.749,E2 5136.749} C_VEL
LIN {X 0,Y 515.503,Z 1129.268,A -85,B 0,C 180,E1 5140.593,E2 5140.593} C_VEL
LIN {X 0,Y 516.082,Z 1113.747,A -85,B 0,C 180,E1 5144.822,E2 5144.822} C_VEL
LIN {X 0,Y 517.205,Z 1093.501,A -85,B 0,C 180,E1 5148.785,E2 5148.785} C_VEL
LIN {X 0,Y 518.87,Z 1067.815,A -85,B 0,C 180,E1 5152.561,E2 5152.561} C_VEL
LIN {X 0,Y 521.178,Z 1037.437,A -85,B 0,C 180,E1 5155.95,E2 5155.95} C_VEL
LIN {X 0,Y 523.697,Z 1003.815,A -85,B 0,C 180,E1 5158.78,E2 5158.78} C_VEL
LIN {X 0,Y 526.168,Z 967.401,A -85,B 0,C 180,E1 5161.025,E2 5161.025} C_VEL
LIN {X 0,Y 528.17,Z 931.07,A -85,B 0,C 180,E1 5162.573,E2 5162.573} C_VEL
LIN {X 0,Y 529.431,Z 893.505,A -85,B 0,C 180,E1 5163.558,E2 5163.558} C_VEL
LIN {X 0,Y 529.023,Z 874.822,A -85,B 0,C 180,E1 5163.912,E2 5163.912} C_VEL
LIN {X 0,Y 514.481,Z 843.44,A -85,B 0,C 180,E1 5165.669,E2 5165.669} C_VEL
LIN {X 0,Y 514.467,Z 843.44,A -85,B 0,C 180,E1 5170.351,E2 5170.351} C_VEL
LIN {X 0,Y 514.44,Z 843.44,A -85,B 0,C 180,E1 5175.067,E2 5175.067} C_VEL
LIN {X 0,Y 514.482,Z 843.44,A -85,B 0,C 180,E1 5179.922,E2 5179.922} C_VEL
LIN {X 0,Y 514.382,Z 843.44,A -85,B 0,C 180,E1 5186,E2 5186} C_VEL
LIN {X 0,Y 514.53,Z 843.44,A -85,B 0,C 180,E1 5191.983,E2 5191.983} C_VEL
LIN {X 0,Y 514.678,Z 843.44,A -85,B 0,C 180,E1 5197.518,E2 5197.518} C_VEL
LIN {X 0,Y 514.814,Z 843.44,A -85,B 0,C 180,E1 5202.899,E2 5202.899} C_VEL
LIN {X 0,Y 514.849,Z 843.44,A -85,B 0,C 180,E1 5208.122,E2 5208.122} C_VEL
LIN {X 0,Y 514.897,Z 843.44,A -85,B 0,C 180,E1 5213.247,E2 5213.247} C_VEL
LIN {X 0,Y 514.971,Z 843.44,A -85,B 0,C 180,E1 5218.518,E2 5218.518} C_VEL
LIN {X 0,Y 514.978,Z 843.44,A -85,B 0,C 180,E1 5223.372,E2 5223.372} C_VEL
LIN {X 0,Y 514.846,Z 843.44,A -85,B 0,C 180,E1 5228.456,E2 5228.456} C_VEL
LIN {X 0,Y 514.755,Z 843.44,A -85,B 0,C 180,E1 5233.911,E2 5233.911} C_VEL
LIN {X 0,Y 514.669,Z 843.44,A -85,B 0,C 180,E1 5239.71,E2 5239.71} C_VEL
LIN {X 0,Y 514.662,Z 843.44,A -85,B 0,C 180,E1 5244.321,E2 5244.321} C_VEL
LIN {X 0,Y 514.463,Z 843.44,A -85,B 0,C 180,E1 5250.019,E2 5250.019} C_VEL
LIN {X 0,Y 514.418,Z 843.44,A -85,B 0,C 180,E1 5256.279,E2 5256.279} C_VEL
LIN {X 0,Y 513.125,Z 843.44,A -85,B 0,C 180,E1 5257.241,E2 5257.241} C_VEL
LIN {X 0,Y 506.493,Z 843.44,A -85,B 0,C 180,E1 5259.863,E2 5259.863} C_VEL
LIN {X 0,Y 506.403,Z 843.44,A -85,B 0,C 180,E1 5260.112,E2 5260.112} C_VEL
LIN {X 0,Y 506.453,Z 843.44,A -85,B 0,C 180,E1 5265.844,E2 5265.844} C_VEL
LIN {X 0,Y 506.55,Z 843.44,A -85,B 0,C 180,E1 5268.466,E2 5268.466} C_VEL
LIN {X 0,Y 513.872,Z 858.794,A -85,B 0,C 180,E1 5269.382,E2 5269.382} C_VEL
LIN {X 0,Y 527.48,Z 883.745,A -85,B 0,C 180,E1 5270.982,E2 5270.982} C_VEL
LIN {X 0,Y 525.876,Z 925.953,A -85,B 0,C 180,E1 5271.997,E2 5271.997} C_VEL
LIN {X 0,Y 523.157,Z 969.078,A -85,B 0,C 180,E1 5273.779,E2 5273.779} C_VEL
LIN {X 0,Y 519.787,Z 1009.392,A -85,B 0,C 180,E1 5276.219,E2 5276.219} C_VEL
LIN {X 0,Y 516.259,Z 1047.397,A -85,B 0,C 180,E1 5279.364,E2 5279.364} C_VEL
LIN {X 0,Y 513.013,Z 1081.633,A -85,B 0,C 180,E1 5283.114,E2 5283.114} C_VEL
LIN {X 0,Y 510.478,Z 1111.033,A -85,B 0,C 180,E1 5287.32,E2 5287.32} C_VEL
LIN {X 0,Y 508.832,Z 1134.143,A -85,B 0,C 180,E1 5291.635,E2 5291.635} C_VEL
LIN {X 0,Y 507.917,Z 1152.301,A -85,B 0,C 180,E1 5296.204,E2 5296.204} C_VEL
LIN {X 0,Y 507.545,Z 1164.58,A -85,B 0,C 180,E1 5300.635,E2 5300.635} C_VEL
LIN {X 0,Y 507.42,Z 1171.905,A -85,B 0,C 180,E1 5304.865,E2 5304.865} C_VEL
LIN {X 0,Y 507.395,Z 1174.657,A -85,B 0,C 180,E1 5308.291,E2 5308.291} C_VEL
LIN {X 0,Y 507.296,Z 1173.627,A -85,B 0,C 180,E1 5313.423,E2 5313.423} C_VEL
LIN {X 0,Y 507.441,Z 1167.916,A -85,B 0,C 180,E1 5317.717,E2 5317.717} C_VEL
LIN {X 0,Y 507.622,Z 1157.768,A -85,B 0,C 180,E1 5322.053,E2 5322.053} C_VEL
LIN {X 0,Y 508.315,Z 1142.486,A -85,B 0,C 180,E1 5326.439,E2 5326.439} C_VEL
LIN {X 0,Y 509.715,Z 1121.372,A -85,B 0,C 180,E1 5330.884,E2 5330.884} C_VEL
LIN {X 0,Y 511.784,Z 1095.247,A -85,B 0,C 180,E1 5335.071,E2 5335.071} C_VEL
LIN {X 0,Y 514.542,Z 1065.168,A -85,B 0,C 180,E1 5338.808,E2 5338.808} C_VEL
LIN {X 0,Y 517.831,Z 1030.973,A -85,B 0,C 180,E1 5342.099,E2 5342.099} C_VEL
LIN {X 0,Y 521.073,Z 994.615,A -85,B 0,C 180,E1 5344.77,E2 5344.77} C_VEL
LIN {X 0,Y 524.231,Z 954.719,A -85,B 0,C 180,E1 5346.898,E2 5346.898} C_VEL
LIN {X 0,Y 526.558,Z 913.248,A -85,B 0,C 180,E1 5348.37,E2 5348.37} C_VEL
LIN {X 0,Y 527.023,Z 882.277,A -85,B 0,C 180,E1 5349.089,E2 5349.089} C_VEL
LIN {X 0,Y 506.596,Z 844.381,A -85,B 0,C 180,E1 5351.48,E2 5351.48} C_VEL
LIN {X 0,Y 506.522,Z 843.44,A -85,B 0,C 180,E1 5351.648,E2 5351.648} C_VEL
LIN {X 0,Y 506.398,Z 843.44,A -85,B 0,C 180,E1 5358.376,E2 5358.376} C_VEL
LIN {X 0,Y 506.639,Z 843.44,A -85,B 0,C 180,E1 5363.797,E2 5363.797} C_VEL
LIN {X 0,Y 506.679,Z 843.44,A -85,B 0,C 180,E1 5370.07,E2 5370.07} C_VEL
LIN {X 0,Y 506.624,Z 843.44,A -85,B 0,C 180,E1 5375.268,E2 5375.268} C_VEL
LIN {X 0,Y 506.559,Z 843.44,A -85,B 0,C 180,E1 5379.158,E2 5379.158} C_VEL
LIN {X 0,Y 512.837,Z 868.98,A -85,B 0,C 180,E1 5379.757,E2 5379.757} C_VEL
LIN {X 0,Y 512.317,Z 900.984,A -85,B 0,C 180,E1 5380.526,E2 5380.526} C_VEL
LIN {X 0,Y 511.362,Z 930.376,A -85,B 0,C 180,E1 5381.91,E2 5381.91} C_VEL
LIN {X 0,Y 510.11,Z 957.729,A -85,B 0,C 180,E1 5383.955,E2 5383.955} C_VEL
LIN {X 0,Y 508.924,Z 980.259,A -85,B 0,C 180,E1 5386.451,E2 5386.451} C_VEL
LIN {X 0,Y 508.059,Z 1000.53,A -85,B 0,C 180,E1 5389.7,E2 5389.7} C_VEL
LIN {X 0,Y 507.612,Z 1014.514,A -85,B 0,C 180,E1 5393.148,E2 5393.148} C_VEL
LIN {X 0,Y 507.47,Z 1022.469,A -85,B 0,C 180,E1 5396.579,E2 5396.579} C_VEL
LIN {X 0,Y 507.511,Z 1024.998,A -85,B 0,C 180,E1 5399.999,E2 5399.999} C_VEL
LIN {X 0,Y 507.474,Z 1022.335,A -85,B 0,C 180,E1 5403.42,E2 5403.42} C_VEL
LIN {X 0,Y 507.626,Z 1014.324,A -85,B 0,C 180,E1 5406.851,E2 5406.851} C_VEL
LIN {X 0,Y 508.085,Z 1000.081,A -85,B 0,C 180,E1 5410.298,E2 5410.298} C_VEL
LIN {X 0,Y 508.97,Z 979.519,A -85,B 0,C 180,E1 5413.546,E2 5413.546} C_VEL
LIN {X 0,Y 510.204,Z 956.589,A -85,B 0,C 180,E1 5416.041,E2 5416.041} C_VEL
LIN {X 0,Y 511.439,Z 929.65,A -85,B 0,C 180,E1 5418.038,E2 5418.038} C_VEL
LIN {X 0,Y 512.436,Z 899.247,A -85,B 0,C 180,E1 5419.459,E2 5419.459} C_VEL
LIN {X 0,Y 512.903,Z 866.79,A -85,B 0,C 180,E1 5420.226,E2 5420.226} C_VEL
LIN {X 0,Y 506.677,Z 843.44,A -85,B 0,C 180,E1 5420.849,E2 5420.849} C_VEL
LIN {X 0,Y 506.588,Z 843.44,A -85,B 0,C 180,E1 5426.632,E2 5426.632} C_VEL
LIN {X 0,Y 506.567,Z 843.44,A -85,B 0,C 180,E1 5432.543,E2 5432.543} C_VEL
LIN {X 0,Y 506.587,Z 843.44,A -85,B 0,C 180,E1 5436.704,E2 5436.704} C_VEL
LIN {X 0,Y 506.38,Z 843.44,A -85,B 0,C 180,E1 5441.622,E2 5441.622} C_VEL
LIN {X 0,Y 506.386,Z 843.44,A -85,B 0,C 180,E1 5448.367,E2 5448.367} C_VEL
LIN {X 0,Y 506.696,Z 844.229,A -85,B 0,C 180,E1 5453.568,E2 5453.568} C_VEL
LIN {X 0,Y 522.809,Z 877.94,A -85,B 0,C 180,E1 5455.589,E2 5455.589} C_VEL
LIN {X 0,Y 521.879,Z 921.419,A -85,B 0,C 180,E1 5456.546,E2 5456.546} C_VEL
LIN {X 0,Y 519.863,Z 959.877,A -85,B 0,C 180,E1 5458.051,E2 5458.051} C_VEL
LIN {X 0,Y 517.293,Z 996.202,A -85,B 0,C 180,E1 5460.158,E2 5460.158} C_VEL
LIN {X 0,Y 514.406,Z 1031.364,A -85,B 0,C 180,E1 5462.973,E2 5462.973} C_VEL
LIN {X 0,Y 511.73,Z 1063.242,A -85,B 0,C 180,E1 5466.415,E2 5466.415} C_VEL
LIN {X 0,Y 509.686,Z 1090.052,A -85,B 0,C 180,E1 5470.251,E2 5470.251} C_VEL
LIN {X 0,Y 508.418,Z 1109.995,A -85,B 0,C 180,E1 5474.009,E2 5474.009} C_VEL
LIN {X 0,Y 507.701,Z 1125.554,A -85,B 0,C 180,E1 5477.949,E2 5477.949} C_VEL
LIN {X 0,Y 507.461,Z 1137.136,A -85,B 0,C 180,E1 5482.283,E2 5482.283} C_VEL
LIN {X 0,Y 507.297,Z 1143.443,A -85,B 0,C 180,E1 5486.577,E2 5486.577} C_VEL
LIN {X 0,Y 507.309,Z 1144.995,A -85,B 0,C 180,E1 5489.999,E2 5489.999} C_VEL
LIN {X 0,Y 507.328,Z 1143.354,A -85,B 0,C 180,E1 5493.421,E2 5493.421} C_VEL
LIN {X 0,Y 507.453,Z 1136.94,A -85,B 0,C 180,E1 5497.716,E2 5497.716} C_VEL
LIN {X 0,Y 507.806,Z 1125.242,A -85,B 0,C 180,E1 5502.047,E2 5502.047} C_VEL
LIN {X 0,Y 508.654,Z 1107.52,A -85,B 0,C 180,E1 5506.426,E2 5506.426} C_VEL
LIN {X 0,Y 510.055,Z 1085.363,A -85,B 0,C 180,E1 5510.414,E2 5510.414} C_VEL
LIN {X 0,Y 512.232,Z 1057.704,A -85,B 0,C 180,E1 5514.16,E2 5514.16} C_VEL
LIN {X 0,Y 514.78,Z 1026.646,A -85,B 0,C 180,E1 5517.359,E2 5517.359} C_VEL
LIN {X 0,Y 517.456,Z 992.984,A -85,B 0,C 180,E1 5519.97,E2 5519.97} C_VEL
LIN {X 0,Y 519.963,Z 956.166,A -85,B 0,C 180,E1 5522.039,E2 5522.039} C_VEL
LIN {X 0,Y 522.023,Z 918.615,A -85,B 0,C 180,E1 5523.441,E2 5523.441} C_VEL
LIN {X 0,Y 522.378,Z 877.2,A -85,B 0,C 180,E1 5524.365,E2 5524.365} C_VEL
LIN {X 0,Y 507.911,Z 847.853,A -85,B 0,C 180,E1 5526.156,E2 5526.156} C_VEL
LIN {X 0,Y 506.553,Z 843.44,A -85,B 0,C 180,E1 5526.428,E2 5526.428} C_VEL
LIN {X 0,Y 506.472,Z 843.44,A -85,B 0,C 180,E1 5531.644,E2 5531.644} C_VEL
LIN {X 0,Y 506.494,Z 843.44,A -85,B 0,C 180,E1 5538.361,E2 5538.361} C_VEL
LIN {X 0,Y 506.509,Z 843.44,A -85,B 0,C 180,E1 5543.815,E2 5543.815} C_VEL
LIN {X 0,Y 506.558,Z 843.44,A -85,B 0,C 180,E1 5550.09,E2 5550.09} C_VEL
LIN {X 0,Y 506.704,Z 843.44,A -85,B 0,C 180,E1 5555.274,E2 5555.274} C_VEL
LIN {X 0,Y 506.866,Z 843.44,A -85,B 0,C 180,E1 5560.82,E2 5560.82} C_VEL
LIN {X 0,Y 507.003,Z 843.44,A -85,B 0,C 180,E1 5566.18,E2 5566.18} C_VEL
LIN {X 0,Y 507.049,Z 843.44,A -85,B 0,C 180,E1 5571.415,E2 5571.415} C_VEL
LIN {X 0,Y 507.204,Z 843.44,A -85,B 0,C 180,E1 5576.578,E2 5576.578} C_VEL
LIN {X 0,Y 507.311,Z 843.44,A -85,B 0,C 180,E1 5581.711,E2 5581.711} C_VEL
LIN {X 0,Y 507.114,Z 843.44,A -85,B 0,C 180,E1 5586.859,E2 5586.859} C_VEL
LIN {X 0,Y 506.898,Z 843.44,A -85,B 0,C 180,E1 5592.069,E2 5592.069} C_VEL
LIN {X 0,Y 506.802,Z 843.44,A -85,B 0,C 180,E1 5597.382,E2 5597.382} C_VEL
LIN {X 0,Y 506.754,Z 843.44,A -85,B 0,C 180,E1 5602.855,E2 5602.855} C_VEL
LIN {X 0,Y 506.558,Z 843.44,A -85,B 0,C 180,E1 5608.568,E2 5608.568} C_VEL
LIN {X 0,Y 506.489,Z 843.44,A -85,B 0,C 180,E1 5614.607,E2 5614.607} C_VEL
LIN {X 0,Y 506.403,Z 843.44,A -85,B 0,C 180,E1 5620.112,E2 5620.112} C_VEL
LIN {X 0,Y 503.91,Z 843.44,A -85,B 0,C 180,E1 5621.572,E2 5621.572} C_VEL
LIN {X 0,Y 498.649,Z 843.44,A -85,B 0,C 180,E1 5623.762,E2 5623.762} C_VEL
LIN {X 0,Y 498.563,Z 843.44,A -85,B 0,C 180,E1 5624.015,E2 5624.015} C_VEL
LIN {X 0,Y 498.569,Z 843.44,A -85,B 0,C 180,E1 5627.776,E2 5627.776} C_VEL
LIN {X 0,Y 507.211,Z 861.491,A -85,B 0,C 180,E1 5628.874,E2 5628.874} C_VEL
LIN {X 0,Y 521.283,Z 886.554,A -85,B 0,C 180,E1 5630.486,E2 5630.486} C_VEL
LIN {X 0,Y 519.526,Z 927.516,A -85,B 0,C 180,E1 5631.511,E2 5631.511} C_VEL
LIN {X 0,Y 516.688,Z 969.195,A -85,B 0,C 180,E1 5633.259,E2 5633.259} C_VEL
LIN {X 0,Y 513.097,Z 1009.277,A -85,B 0,C 180,E1 5635.708,E2 5635.708} C_VEL
LIN {X 0,Y 509.261,Z 1047.404,A -85,B 0,C 180,E1 5638.898,E2 5638.898} C_VEL
LIN {X 0,Y 505.8,Z 1080.812,A -85,B 0,C 180,E1 5642.586,E2 5642.586} C_VEL
LIN {X 0,Y 502.854,Z 1111.035,A -85,B 0,C 180,E1 5646.957,E2 5646.957} C_VEL
LIN {X 0,Y 501.023,Z 1135.293,A -85,B 0,C 180,E1 5651.604,E2 5651.604} C_VEL
LIN {X 0,Y 500.035,Z 1153.747,A -85,B 0,C 180,E1 5656.428,E2 5656.428} C_VEL
LIN {X 0,Y 499.573,Z 1166.332,A -85,B 0,C 180,E1 5661.284,E2 5661.284} C_VEL
LIN {X 0,Y 499.526,Z 1171.905,A -85,B 0,C 180,E1 5664.783,E2 5664.783} C_VEL
LIN {X 0,Y 499.496,Z 1174.657,A -85,B 0,C 180,E1 5668.264,E2 5668.264} C_VEL
LIN {X 0,Y 499.383,Z 1174.657,A -85,B 0,C 180,E1 5671.738,E2 5671.738} C_VEL
LIN {X 0,Y 499.495,Z 1170.702,A -85,B 0,C 180,E1 5676.091,E2 5676.091} C_VEL
LIN {X 0,Y 499.74,Z 1162.434,A -85,B 0,C 180,E1 5680.475,E2 5680.475} C_VEL
LIN {X 0,Y 500.293,Z 1147.474,A -85,B 0,C 180,E1 5685.414,E2 5685.414} C_VEL
LIN {X 0,Y 501.511,Z 1127.397,A -85,B 0,C 180,E1 5690.066,E2 5690.066} C_VEL
LIN {X 0,Y 503.781,Z 1101.462,A -85,B 0,C 180,E1 5694.56,E2 5694.56} C_VEL
LIN {X 0,Y 506.975,Z 1069.525,A -85,B 0,C 180,E1 5698.771,E2 5698.771} C_VEL
LIN {X 0,Y 510.718,Z 1033.44,A -85,B 0,C 180,E1 5702.376,E2 5702.376} C_VEL
LIN {X 0,Y 514.282,Z 996.481,A -85,B 0,C 180,E1 5705.167,E2 5705.167} C_VEL
LIN {X 0,Y 517.719,Z 956.151,A -85,B 0,C 180,E1 5707.364,E2 5707.364} C_VEL
LIN {X 0,Y 520.255,Z 914.852,A -85,B 0,C 180,E1 5708.867,E2 5708.867} C_VEL
LIN {X 0,Y 521.034,Z 885.707,A -85,B 0,C 180,E1 5709.554,E2 5709.554} C_VEL
LIN {X 0,Y 498.578,Z 844.404,A -85,B 0,C 180,E1 5712.185,E2 5712.185} C_VEL
LIN {X 0,Y 498.46,Z 843.44,A -85,B 0,C 180,E1 5712.498,E2 5712.498} C_VEL
LIN {X 0,Y 498.448,Z 843.44,A -85,B 0,C 180,E1 5718.07,E2 5718.07} C_VEL
LIN {X 0,Y 498.697,Z 843.44,A -85,B 0,C 180,E1 5724.773,E2 5724.773} C_VEL
LIN {X 0,Y 498.712,Z 843.44,A -85,B 0,C 180,E1 5730.94,E2 5730.94} C_VEL
LIN {X 0,Y 498.655,Z 843.44,A -85,B 0,C 180,E1 5736.753,E2 5736.753} C_VEL
LIN {X 0,Y 498.651,Z 844.034,A -85,B 0,C 180,E1 5738.92,E2 5738.92} C_VEL
LIN {X 0,Y 505.24,Z 869.393,A -85,B 0,C 180,E1 5739.514,E2 5739.514} C_VEL
LIN {X 0,Y 504.793,Z 901.141,A -85,B 0,C 180,E1 5740.256,E2 5740.256} C_VEL
LIN {X 0,Y 503.839,Z 931.014,A -85,B 0,C 180,E1 5741.647,E2 5741.647} C_VEL
LIN {X 0,Y 502.586,Z 958.604,A -85,B 0,C 180,E1 5743.708,E2 5743.708} C_VEL
LIN {X 0,Y 501.335,Z 981.459,A -85,B 0,C 180,E1 5746.242,E2 5746.242} C_VEL
LIN {X 0,Y 500.388,Z 1000.688,A -85,B 0,C 180,E1 5749.387,E2 5749.387} C_VEL
LIN {X 0,Y 499.854,Z 1013.572,A -85,B 0,C 180,E1 5752.603,E2 5752.603} C_VEL
LIN {X 0,Y 499.627,Z 1021.022,A -85,B 0,C 180,E1 5755.655,E2 5755.655} C_VEL
LIN {X 0,Y 499.546,Z 1024.376,A -85,B 0,C 180,E1 5758.262,E2 5758.262} C_VEL
LIN {X 0,Y 499.544,Z 1024.305,A -85,B 0,C 180,E1 5761.736,E2 5761.736} C_VEL
LIN {X 0,Y 499.631,Z 1019.061,A -85,B 0,C 180,E1 5765.215,E2 5765.215} C_VEL
LIN {X 0,Y 500.003,Z 1008.516,A -85,B 0,C 180,E1 5768.707,E2 5768.707} C_VEL
LIN {X 0,Y 500.709,Z 992.371,A -85,B 0,C 180,E1 5771.997,E2 5771.997} C_VEL
LIN {X 0,Y 501.854,Z 971.083,A -85,B 0,C 180,E1 5774.895,E2 5774.895} C_VEL
LIN {X 0,Y 503.139,Z 946.751,A -85,B 0,C 180,E1 5777.172,E2 5777.172} C_VEL
LIN {X 0,Y 504.368,Z 918.022,A -85,B 0,C 180,E1 5778.966,E2 5778.966} C_VEL
LIN {X 0,Y 505.229,Z 886.798,A -85,B 0,C 180,E1 5780.117,E2 5780.117} C_VEL
LIN {X 0,Y 504.493,Z 863.477,A -85,B 0,C 180,E1 5780.586,E2 5780.586} C_VEL
LIN {X 0,Y 498.744,Z 843.44,A -85,B 0,C 180,E1 5781.173,E2 5781.173} C_VEL
LIN {X 0,Y 498.618,Z 843.44,A -85,B 0,C 180,E1 5787.092,E2 5787.092} C_VEL
LIN {X 0,Y 498.676,Z 843.44,A -85,B 0,C 180,E1 5793.124,E2 5793.124} C_VEL
LIN {X 0,Y 498.502,Z 843.44,A -85,B 0,C 180,E1 5799.624,E2 5799.624} C_VEL
LIN {X 0,Y 498.376,Z 843.44,A -85,B 0,C 180,E1 5805.67,E2 5805.67} C_VEL
LIN {X 0,Y 498.612,Z 843.44,A -85,B 0,C 180,E1 5812.132,E2 5812.132} C_VEL
LIN {X 0,Y 498.707,Z 844.315,A -85,B 0,C 180,E1 5812.777,E2 5812.777} C_VEL
LIN {X 0,Y 515.001,Z 877.141,A -85,B 0,C 180,E1 5814.935,E2 5814.935} C_VEL
LIN {X 0,Y 516.405,Z 883.302,A -85,B 0,C 180,E1 5815.171,E2 5815.171} C_VEL
LIN {X 0,Y 514.985,Z 926.957,A -85,B 0,C 180,E1 5816.235,E2 5816.235} C_VEL
LIN {X 0,Y 512.628,Z 965.893,A -85,B 0,C 180,E1 5817.881,E2 5817.881} C_VEL
LIN {X 0,Y 509.735,Z 1002.535,A -85,B 0,C 180,E1 5820.161,E2 5820.161} C_VEL
LIN {X 0,Y 506.764,Z 1036.026,A -85,B 0,C 180,E1 5823.016,E2 5823.016} C_VEL
LIN {X 0,Y 504.069,Z 1065.468,A -85,B 0,C 180,E1 5826.333,E2 5826.333} C_VEL
LIN {X 0,Y 501.915,Z 1091.744,A -85,B 0,C 180,E1 5830.226,E2 5830.226} C_VEL
LIN {X 0,Y 500.577,Z 1111.951,A -85,B 0,C 180,E1 5834.202,E2 5834.202} C_VEL
LIN {X 0,Y 499.825,Z 1126.911,A -85,B 0,C 180,E1 5838.2,E2 5838.2} C_VEL
LIN {X 0,Y 499.573,Z 1137.135,A -85,B 0,C 180,E1 5842.16,E2 5842.16} C_VEL
LIN {X 0,Y 499.392,Z 1143.442,A -85,B 0,C 180,E1 5846.523,E2 5846.523} C_VEL
LIN {X 0,Y 499.43,Z 1144.995,A -85,B 0,C 180,E1 5849.999,E2 5849.999} C_VEL
LIN {X 0,Y 499.427,Z 1143.355,A -85,B 0,C 180,E1 5853.475,E2 5853.475} C_VEL
LIN {X 0,Y 499.583,Z 1136.942,A -85,B 0,C 180,E1 5857.838,E2 5857.838} C_VEL
LIN {X 0,Y 499.964,Z 1125.244,A -85,B 0,C 180,E1 5862.238,E2 5862.238} C_VEL
LIN {X 0,Y 500.912,Z 1107.522,A -85,B 0,C 180,E1 5866.687,E2 5866.687} C_VEL
LIN {X 0,Y 502.495,Z 1084.94,A -85,B 0,C 180,E1 5870.802,E2 5870.802} C_VEL
LIN {X 0,Y 504.869,Z 1057.348,A -85,B 0,C 180,E1 5874.58,E2 5874.58} C_VEL
LIN {X 0,Y 507.611,Z 1026.651,A -85,B 0,C 180,E1 5877.779,E2 5877.779} C_VEL
LIN {X 0,Y 510.526,Z 992.923,A -85,B 0,C 180,E1 5880.424,E2 5880.424} C_VEL
LIN {X 0,Y 513.202,Z 956.18,A -85,B 0,C 180,E1 5882.513,E2 5882.513} C_VEL
LIN {X 0,Y 515.478,Z 917.386,A -85,B 0,C 180,E1 5883.963,E2 5883.963} C_VEL
LIN {X 0,Y 516.246,Z 880.43,A -85,B 0,C 180,E1 5884.804,E2 5884.804} C_VEL
LIN {X 0,Y 501.074,Z 849.142,A -85,B 0,C 180,E1 5886.799,E2 5886.799} C_VEL
LIN {X 0,Y 498.585,Z 843.44,A -85,B 0,C 180,E1 5887.219,E2 5887.219} C_VEL
LIN {X 0,Y 498.56,Z 843.44,A -85,B 0,C 180,E1 5893.216,E2 5893.216} C_VEL
LIN {X 0,Y 498.51,Z 843.44,A -85,B 0,C 180,E1 5899.404,E2 5899.404} C_VEL
LIN {X 0,Y 498.553,Z 843.44,A -85,B 0,C 180,E1 5905.084,E2 5905.084} C_VEL
LIN {X 0,Y 498.633,Z 843.44,A -85,B 0,C 180,E1 5911.714,E2 5911.714} C_VEL
LIN {X 0,Y 498.802,Z 843.44,A -85,B 0,C 180,E1 5916.762,E2 5916.762} C_VEL
LIN {X 0,Y 498.961,Z 843.44,A -85,B 0,C 180,E1 5922.338,E2 5922.338} C_VEL
LIN {X 0,Y 499.018,Z 843.44,A -85,B 0,C 180,E1 5927.74,E2 5927.74} C_VEL
LIN {X 0,Y 499.08,Z 843.44,A -85,B 0,C 180,E1 5933.031,E2 5933.031} C_VEL
LIN {X 0,Y 499.196,Z 843.44,A -85,B 0,C 180,E1 5938.263,E2 5938.263} C_VEL
LIN {X 0,Y 499.169,Z 843.44,A -85,B 0,C 180,E1 5943.478,E2 5943.478} C_VEL
LIN {X 0,Y 499.041,Z 843.44,A -85,B 0,C 180,E1 5948.725,E2 5948.725} C_VEL
LIN {X 0,Y 498.959,Z 843.44,A -85,B 0,C 180,E1 5954.049,E2 5954.049} C_VEL
LIN {X 0,Y 498.811,Z 843.44,A -85,B 0,C 180,E1 5959.782,E2 5959.782} C_VEL
LIN {X 0,Y 498.785,Z 843.44,A -85,B 0,C 180,E1 5965.148,E2 5965.148} C_VEL
LIN {X 0,Y 498.548,Z 843.44,A -85,B 0,C 180,E1 5971.748,E2 5971.748} C_VEL
LIN {X 0,Y 498.534,Z 843.44,A -85,B 0,C 180,E1 5977.847,E2 5977.847} C_VEL
LIN {X 0,Y 498.563,Z 843.44,A -85,B 0,C 180,E1 5984.015,E2 5984.015} C_VEL
LIN {X 0,Y 494.587,Z 843.44,A -85,B 0,C 180,E1 5985.297,E2 5985.297} C_VEL
LIN {X 0,Y 490.657,Z 843.44,A -85,B 0,C 180,E1 5986.601,E2 5986.601} C_VEL
LIN {X 0,Y 490.706,Z 844.249,A -85,B 0,C 180,E1 5987.109,E2 5987.109} C_VEL
LIN {X 0,Y 514.916,Z 890.079,A -85,B 0,C 180,E1 5990.022,E2 5990.022} C_VEL
LIN {X 0,Y 513.215,Z 928.87,A -85,B 0,C 180,E1 5991.008,E2 5991.008} C_VEL
LIN {X 0,Y 510.13,Z 970.523,A -85,B 0,C 180,E1 5992.791,E2 5992.791} C_VEL
LIN {X 0,Y 506.3,Z 1010.436,A -85,B 0,C 180,E1 5995.279,E2 5995.279} C_VEL
LIN {X 0,Y 502.221,Z 1047.749,A -85,B 0,C 180,E1 5998.45,E2 5998.45} C_VEL
LIN {X 0,Y 498.402,Z 1081.565,A -85,B 0,C 180,E1 6002.249,E2 6002.249} C_VEL
LIN {X 0,Y 495.324,Z 1111.037,A -85,B 0,C 180,E1 6006.586,E2 6006.586} C_VEL
LIN {X 0,Y 493.314,Z 1134.846,A -85,B 0,C 180,E1 6011.2,E2 6011.2} C_VEL
LIN {X 0,Y 492.196,Z 1153.747,A -85,B 0,C 180,E1 6016.208,E2 6016.208} C_VEL
LIN {X 0,Y 491.692,Z 1166.331,A -85,B 0,C 180,E1 6021.144,E2 6021.144} C_VEL
LIN {X 0,Y 491.622,Z 1171.905,A -85,B 0,C 180,E1 6024.699,E2 6024.699} C_VEL
LIN {X 0,Y 491.59,Z 1174.657,A -85,B 0,C 180,E1 6028.236,E2 6028.236} C_VEL
LIN {X 0,Y 491.48,Z 1174.657,A -85,B 0,C 180,E1 6031.766,E2 6031.766} C_VEL
LIN {X 0,Y 491.617,Z 1170.702,A -85,B 0,C 180,E1 6036.189,E2 6036.189} C_VEL
LIN {X 0,Y 491.858,Z 1162.433,A -85,B 0,C 180,E1 6040.645,E2 6040.645} C_VEL
LIN {X 0,Y 492.462,Z 1147.674,A -85,B 0,C 180,E1 6045.607,E2 6045.607} C_VEL
LIN {X 0,Y 493.8,Z 1127.746,A -85,B 0,C 180,E1 6050.319,E2 6050.319} C_VEL
LIN {X 0,Y 496.192,Z 1102.687,A -85,B 0,C 180,E1 6054.761,E2 6054.761} C_VEL
LIN {X 0,Y 499.341,Z 1073.005,A -85,B 0,C 180,E1 6058.806,E2 6058.806} C_VEL
LIN {X 0,Y 503.134,Z 1039.314,A -85,B 0,C 180,E1 6062.343,E2 6062.343} C_VEL
LIN {X 0,Y 506.965,Z 1003.286,A -85,B 0,C 180,E1 6065.227,E2 6065.227} C_VEL
LIN {X 0,Y 510.59,Z 964.834,A -85,B 0,C 180,E1 6067.497,E2 6067.497} C_VEL
LIN {X 0,Y 513.424,Z 924.075,A -85,B 0,C 180,E1 6069.156,E2 6069.156} C_VEL
LIN {X 0,Y 514.695,Z 888.652,A -85,B 0,C 180,E1 6070.024,E2 6070.024} C_VEL
LIN {X 0,Y 490.621,Z 844.514,A -85,B 0,C 180,E1 6072.912,E2 6072.912} C_VEL
LIN {X 0,Y 490.524,Z 843.44,A -85,B 0,C 180,E1 6073.106,E2 6073.106} C_VEL
LIN {X 0,Y 490.587,Z 843.44,A -85,B 0,C 180,E1 6079.604,E2 6079.604} C_VEL
LIN {X 0,Y 490.755,Z 843.44,A -85,B 0,C 180,E1 6086.269,E2 6086.269} C_VEL
LIN {X 0,Y 490.769,Z 843.44,A -85,B 0,C 180,E1 6092.436,E2 6092.436} C_VEL
LIN {X 0,Y 490.77,Z 843.44,A -85,B 0,C 180,E1 6098.617,E2 6098.617} C_VEL
LIN {X 0,Y 497.653,Z 872.791,A -85,B 0,C 180,E1 6099.308,E2 6099.308} C_VEL
LIN {X 0,Y 497.187,Z 904.348,A -85,B 0,C 180,E1 6100.088,E2 6100.088} C_VEL
LIN {X 0,Y 496.287,Z 933.218,A -85,B 0,C 180,E1 6101.474,E2 6101.474} C_VEL
LIN {X 0,Y 495.071,Z 959.456,A -85,B 0,C 180,E1 6103.454,E2 6103.454} C_VEL
LIN {X 0,Y 493.734,Z 982.594,A -85,B 0,C 180,E1 6106.026,E2 6106.026} C_VEL
LIN {X 0,Y 492.75,Z 1001.659,A -85,B 0,C 180,E1 6109.152,E2 6109.152} C_VEL
LIN {X 0,Y 492.148,Z 1014.967,A -85,B 0,C 180,E1 6112.487,E2 6112.487} C_VEL
LIN {X 0,Y 491.873,Z 1022.404,A -85,B 0,C 180,E1 6115.586,E2 6115.586} C_VEL
LIN {X 0,Y 491.747,Z 1025.568,A -85,B 0,C 180,E1 6118.235,E2 6118.235} C_VEL
LIN {X 0,Y 491.745,Z 1025.442,A -85,B 0,C 180,E1 6121.763,E2 6121.763} C_VEL
LIN {X 0,Y 491.88,Z 1020.344,A -85,B 0,C 180,E1 6125.297,E2 6125.297} C_VEL
LIN {X 0,Y 492.273,Z 1009.693,A -85,B 0,C 180,E1 6128.845,E2 6128.845} C_VEL
LIN {X 0,Y 493.039,Z 993.399,A -85,B 0,C 180,E1 6132.186,E2 6132.186} C_VEL
LIN {X 0,Y 494.255,Z 971.867,A -85,B 0,C 180,E1 6135.129,E2 6135.129} C_VEL
LIN {X 0,Y 495.611,Z 947.255,A -85,B 0,C 180,E1 6137.441,E2 6137.441} C_VEL
LIN {X 0,Y 496.873,Z 918.732,A -85,B 0,C 180,E1 6139.23,E2 6139.23} C_VEL
LIN {X 0,Y 497.748,Z 887.062,A -85,B 0,C 180,E1 6140.399,E2 6140.399} C_VEL
LIN {X 0,Y 496.94,Z 864.834,A -85,B 0,C 180,E1 6140.854,E2 6140.854} C_VEL
LIN {X 0,Y 490.856,Z 843.44,A -85,B 0,C 180,E1 6141.466,E2 6141.466} C_VEL
LIN {X 0,Y 490.68,Z 843.44,A -85,B 0,C 180,E1 6147.568,E2 6147.568} C_VEL
LIN {X 0,Y 490.729,Z 843.44,A -85,B 0,C 180,E1 6153.731,E2 6153.731} C_VEL
LIN {X 0,Y 490.561,Z 843.44,A -85,B 0,C 180,E1 6160.397,E2 6160.397} C_VEL
LIN {X 0,Y 490.485,Z 843.44,A -85,B 0,C 180,E1 6167.222,E2 6167.222} C_VEL
LIN {X 0,Y 490.747,Z 844.228,A -85,B 0,C 180,E1 6171.941,E2 6171.941} C_VEL
LIN {X 0,Y 507.328,Z 876.269,A -85,B 0,C 180,E1 6174.207,E2 6174.207} C_VEL
LIN {X 0,Y 510.274,Z 884.228,A -85,B 0,C 180,E1 6174.626,E2 6174.626} C_VEL
LIN {X 0,Y 508.738,Z 926.217,A -85,B 0,C 180,E1 6175.674,E2 6175.674} C_VEL
LIN {X 0,Y 506.063,Z 963.988,A -85,B 0,C 180,E1 6177.301,E2 6177.301} C_VEL
LIN {X 0,Y 503.085,Z 999.444,A -85,B 0,C 180,E1 6179.476,E2 6179.476} C_VEL
LIN {X 0,Y 499.721,Z 1034.066,A -85,B 0,C 180,E1 6182.397,E2 6182.397} C_VEL
LIN {X 0,Y 496.795,Z 1064.008,A -85,B 0,C 180,E1 6185.766,E2 6185.766} C_VEL
LIN {X 0,Y 494.391,Z 1089.94,A -85,B 0,C 180,E1 6189.595,E2 6189.595} C_VEL
LIN {X 0,Y 492.898,Z 1109.99,A -85,B 0,C 180,E1 6193.491,E2 6193.491} C_VEL
LIN {X 0,Y 492.012,Z 1125.548,A -85,B 0,C 180,E1 6197.559,E2 6197.559} C_VEL
LIN {X 0,Y 491.679,Z 1137.133,A -85,B 0,C 180,E1 6202.034,E2 6202.034} C_VEL
LIN {X 0,Y 491.488,Z 1143.442,A -85,B 0,C 180,E1 6206.467,E2 6206.467} C_VEL
LIN {X 0,Y 491.53,Z 1144.995,A -85,B 0,C 180,E1 6209.999,E2 6209.999} C_VEL
LIN {X 0,Y 491.525,Z 1143.356,A -85,B 0,C 180,E1 6213.531,E2 6213.531} C_VEL
LIN {X 0,Y 491.704,Z 1136.944,A -85,B 0,C 180,E1 6217.964,E2 6217.964} C_VEL
LIN {X 0,Y 492.127,Z 1125.246,A -85,B 0,C 180,E1 6222.436,E2 6222.436} C_VEL
LIN {X 0,Y 493.146,Z 1107.525,A -85,B 0,C 180,E1 6226.958,E2 6226.958} C_VEL
LIN {X 0,Y 494.909,Z 1084.943,A -85,B 0,C 180,E1 6231.136,E2 6231.136} C_VEL
LIN {X 0,Y 497.36,Z 1058.546,A -85,B 0,C 180,E1 6234.827,E2 6234.827} C_VEL
LIN {X 0,Y 500.395,Z 1027.08,A -85,B 0,C 180,E1 6238.174,E2 6238.174} C_VEL
LIN {X 0,Y 503.611,Z 992.932,A -85,B 0,C 180,E1 6240.887,E2 6240.887} C_VEL
LIN {X 0,Y 506.666,Z 954.318,A -85,B 0,C 180,E1 6243.105,E2 6243.105} C_VEL
LIN {X 0,Y 509.322,Z 914.359,A -85,B 0,C 180,E1 6244.607,E2 6244.607} C_VEL
LIN {X 0,Y 509.864,Z 882.567,A -85,B 0,C 180,E1 6245.352,E2 6245.352} C_VEL
LIN {X 0,Y 496.133,Z 854.387,A -85,B 0,C 180,E1 6247.207,E2 6247.207} C_VEL
LIN {X 0,Y 490.708,Z 844.298,A -85,B 0,C 180,E1 6247.952,E2 6247.952} C_VEL
LIN {X 0,Y 490.625,Z 843.44,A -85,B 0,C 180,E1 6248.113,E2 6248.113} C_VEL
LIN {X 0,Y 490.652,Z 843.44,A -85,B 0,C 180,E1 6252.758,E2 6252.758} C_VEL
LIN {X 0,Y 490.671,Z 843.44,A -85,B 0,C 180,E1 6257.782,E2 6257.782} C_VEL
LIN {X 0,Y 490.56,Z 843.44,A -85,B 0,C 180,E1 6264.101,E2 6264.101} C_VEL
LIN {X 0,Y 490.648,Z 843.44,A -85,B 0,C 180,E1 6270.417,E2 6270.417} C_VEL
LIN {X 0,Y 490.874,Z 843.44,A -85,B 0,C 180,E1 6276.364,E2 6276.364} C_VEL
LIN {X 0,Y 491.032,Z 843.44,A -85,B 0,C 180,E1 6282.043,E2 6282.043} C_VEL
LIN {X 0,Y 491.11,Z 843.44,A -85,B 0,C 180,E1 6287.539,E2 6287.539} C_VEL
LIN {X 0,Y 491.17,Z 843.44,A -85,B 0,C 180,E1 6292.919,E2 6292.919} C_VEL
LIN {X 0,Y 491.296,Z 843.44,A -85,B 0,C 180,E1 6298.235,E2 6298.235} C_VEL
LIN {X 0,Y 491.263,Z 843.44,A -85,B 0,C 180,E1 6303.534,E2 6303.534} C_VEL
LIN {X 0,Y 491.097,Z 843.44,A -85,B 0,C 180,E1 6309.39,E2 6309.39} C_VEL
LIN {X 0,Y 491.026,Z 843.44,A -85,B 0,C 180,E1 6314.281,E2 6314.281} C_VEL
LIN {X 0,Y 490.908,Z 843.44,A -85,B 0,C 180,E1 6319.831,E2 6319.831} C_VEL
LIN {X 0,Y 490.813,Z 843.44,A -85,B 0,C 180,E1 6325.585,E2 6325.585} C_VEL
LIN {X 0,Y 490.672,Z 843.44,A -85,B 0,C 180,E1 6331.637,E2 6331.637} C_VEL
LIN {X 0,Y 490.605,Z 843.44,A -85,B 0,C 180,E1 6338.111,E2 6338.111} C_VEL
LIN {X 0,Y 490.589,Z 843.44,A -85,B 0,C 180,E1 6344.017,E2 6344.017} C_VEL
LIN {X 0,Y 490.657,Z 843.44,A -85,B 0,C 180,E1 6346.601,E2 6346.601} C_VEL
LIN {X 0,Y 491.626,Z 846.105,A -85,B 0,C 180,E1 6347.165,E2 6347.165} C_VEL
LIN {X 0,Y 494.243,Z 855.581,A -85,B 0,C 180,E1 6347.637,E2 6347.637} C_VEL
LIN {X 0,Y 497.359,Z 872.237,A -85,B 0,C 180,E1 6348.211,E2 6348.211} C_VEL
LIN {X 0,Y 498.405,Z 874.201,A -85,B 0,C 180,E1 6348.339,E2 6348.339} C_VEL
LIN {X 0,Y 508.407,Z 892.166,A -85,B 0,C 180,E1 6349.538,E2 6349.538} C_VEL
LIN {X 0,Y 506.473,Z 932.622,A -85,B 0,C 180,E1 6350.63,E2 6350.63} C_VEL
LIN {X 0,Y 503.453,Z 973.156,A -85,B 0,C 180,E1 6352.383,E2 6352.383} C_VEL
LIN {X 0,Y 499.52,Z 1011.572,A -85,B 0,C 180,E1 6354.837,E2 6354.837} C_VEL
LIN {X 0,Y 495.113,Z 1048.551,A -85,B 0,C 180,E1 6358.034,E2 6358.034} C_VEL
LIN {X 0,Y 491.035,Z 1082.257,A -85,B 0,C 180,E1 6361.894,E2 6361.894} C_VEL
LIN {X 0,Y 487.809,Z 1111.039,A -85,B 0,C 180,E1 6366.203,E2 6366.203} C_VEL
LIN {X 0,Y 485.526,Z 1134.848,A -85,B 0,C 180,E1 6370.887,E2 6370.887} C_VEL
LIN {X 0,Y 484.394,Z 1152.806,A -85,B 0,C 180,E1 6375.673,E2 6375.673} C_VEL
LIN {X 0,Y 483.903,Z 1165.216,A -85,B 0,C 180,E1 6380.473,E2 6380.473} C_VEL
LIN {X 0,Y 483.721,Z 1171.905,A -85,B 0,C 180,E1 6384.613,E2 6384.613} C_VEL
LIN {X 0,Y 483.714,Z 1174.657,A -85,B 0,C 180,E1 6388.207,E2 6388.207} C_VEL
LIN {X 0,Y 483.577,Z 1174.657,A -85,B 0,C 180,E1 6391.795,E2 6391.795} C_VEL
LIN {X 0,Y 483.73,Z 1170.702,A -85,B 0,C 180,E1 6396.29,E2 6396.29} C_VEL
LIN {X 0,Y 483.97,Z 1162.433,A -85,B 0,C 180,E1 6400.82,E2 6400.82} C_VEL
LIN {X 0,Y 484.66,Z 1147.675,A -85,B 0,C 180,E1 6405.865,E2 6405.865} C_VEL
LIN {X 0,Y 486.251,Z 1127.059,A -85,B 0,C 180,E1 6410.798,E2 6410.798} C_VEL
LIN {X 0,Y 488.922,Z 1100.921,A -85,B 0,C 180,E1 6415.449,E2 6415.449} C_VEL
LIN {X 0,Y 492.563,Z 1069.903,A -85,B 0,C 180,E1 6419.648,E2 6419.648} C_VEL
LIN {X 0,Y 496.989,Z 1033.517,A -85,B 0,C 180,E1 6423.379,E2 6423.379} C_VEL
LIN {X 0,Y 501.169,Z 996.422,A -85,B 0,C 180,E1 6426.234,E2 6426.234} C_VEL
LIN {X 0,Y 504.677,Z 959.214,A -85,B 0,C 180,E1 6428.297,E2 6428.297} C_VEL
LIN {X 0,Y 507.224,Z 919.582,A -85,B 0,C 180,E1 6429.79,E2 6429.79} C_VEL
LIN {X 0,Y 508.166,Z 891.347,A -85,B 0,C 180,E1 6430.499,E2 6430.499} C_VEL
LIN {X 0,Y 482.668,Z 844.594,A -85,B 0,C 180,E1 6433.656,E2 6433.656} C_VEL
LIN {X 0,Y 482.555,Z 843.44,A -85,B 0,C 180,E1 6433.813,E2 6433.813} C_VEL
LIN {X 0,Y 482.629,Z 843.44,A -85,B 0,C 180,E1 6438.847,E2 6438.847} C_VEL
LIN {X 0,Y 482.774,Z 843.44,A -85,B 0,C 180,E1 6444.633,E2 6444.633} C_VEL
LIN {X 0,Y 482.856,Z 843.44,A -85,B 0,C 180,E1 6449.889,E2 6449.889} C_VEL
LIN {X 0,Y 482.807,Z 843.44,A -85,B 0,C 180,E1 6455.942,E2 6455.942} C_VEL
LIN {X 0,Y 482.861,Z 844.191,A -85,B 0,C 180,E1 6458.348,E2 6458.348} C_VEL
LIN {X 0,Y 490.06,Z 872.343,A -85,B 0,C 180,E1 6459.04,E2 6459.04} C_VEL
LIN {X 0,Y 489.659,Z 905.242,A -85,B 0,C 180,E1 6459.833,E2 6459.833} C_VEL
LIN {X 0,Y 488.752,Z 934.936,A -85,B 0,C 180,E1 6461.267,E2 6461.267} C_VEL
LIN {X 0,Y 487.488,Z 961.513,A -85,B 0,C 180,E1 6463.305,E2 6463.305} C_VEL
LIN {X 0,Y 486.154,Z 983.725,A -85,B 0,C 180,E1 6465.803,E2 6465.803} C_VEL
LIN {X 0,Y 485.173,Z 1001.827,A -85,B 0,C 180,E1 6468.753,E2 6468.753} C_VEL
LIN {X 0,Y 484.503,Z 1014.927,A -85,B 0,C 180,E1 6471.916,E2 6471.916} C_VEL
LIN {X 0,Y 484.153,Z 1023.822,A -85,B 0,C 180,E1 6475.516,E2 6475.516} C_VEL
LIN {X 0,Y 484.001,Z 1026.98,A -85,B 0,C 180,E1 6478.207,E2 6478.207} C_VEL
LIN {X 0,Y 483.999,Z 1026.822,A -85,B 0,C 180,E1 6481.792,E2 6481.792} C_VEL
LIN {X 0,Y 484.137,Z 1021.628,A -85,B 0,C 180,E1 6485.382,E2 6485.382} C_VEL
LIN {X 0,Y 484.545,Z 1010.865,A -85,B 0,C 180,E1 6488.987,E2 6488.987} C_VEL
LIN {X 0,Y 485.398,Z 994.392,A -85,B 0,C 180,E1 6492.381,E2 6492.381} C_VEL
LIN {X 0,Y 486.642,Z 973.257,A -85,B 0,C 180,E1 6495.302,E2 6495.302} C_VEL
LIN {X 0,Y 488.102,Z 947.753,A -85,B 0,C 180,E1 6497.718,E2 6497.718} C_VEL
LIN {X 0,Y 489.405,Z 918.776,A -85,B 0,C 180,E1 6499.535,E2 6499.535} C_VEL
LIN {X 0,Y 490.239,Z 887.86,A -85,B 0,C 180,E1 6500.677,E2 6500.677} C_VEL
LIN {X 0,Y 489.814,Z 867.477,A -85,B 0,C 180,E1 6501.094,E2 6501.094} C_VEL
LIN {X 0,Y 482.928,Z 843.44,A -85,B 0,C 180,E1 6501.803,E2 6501.803} C_VEL
LIN {X 0,Y 482.716,Z 843.44,A -85,B 0,C 180,E1 6508.062,E2 6508.062} C_VEL
LIN {X 0,Y 482.739,Z 843.44,A -85,B 0,C 180,E1 6514.367,E2 6514.367} C_VEL
LIN {X 0,Y 482.671,Z 843.44,A -85,B 0,C 180,E1 6518.851,E2 6518.851} C_VEL
LIN {X 0,Y 482.493,Z 843.44,A -85,B 0,C 180,E1 6523.798,E2 6523.798} C_VEL
LIN {X 0,Y 482.734,Z 843.44,A -85,B 0,C 180,E1 6531.036,E2 6531.036} C_VEL
LIN {X 0,Y 485.192,Z 849.127,A -85,B 0,C 180,E1 6531.438,E2 6531.438} C_VEL
LIN {X 0,Y 500.784,Z 877.915,A -85,B 0,C 180,E1 6533.6,E2 6533.6} C_VEL
LIN {X 0,Y 504.178,Z 885.695,A -85,B 0,C 180,E1 6534.077,E2 6534.077} C_VEL
LIN {X 0,Y 502.457,Z 927.615,A -85,B 0,C 180,E1 6535.154,E2 6535.154} C_VEL
LIN {X 0,Y 499.543,Z 965.423,A -85,B 0,C 180,E1 6536.82,E2 6536.82} C_VEL
LIN {X 0,Y 496.008,Z 1000.988,A -85,B 0,C 180,E1 6539.12,E2 6539.12} C_VEL
LIN {X 0,Y 492.588,Z 1033.756,A -85,B 0,C 180,E1 6541.93,E2 6541.93} C_VEL
LIN {X 0,Y 489.474,Z 1063.536,A -85,B 0,C 180,E1 6545.315,E2 6545.315} C_VEL
LIN {X 0,Y 486.826,Z 1089.508,A -85,B 0,C 180,E1 6549.187,E2 6549.187} C_VEL
LIN {X 0,Y 485.189,Z 1109.988,A -85,B 0,C 180,E1 6553.221,E2 6553.221} C_VEL
LIN {X 0,Y 484.113,Z 1126.908,A -85,B 0,C 180,E1 6557.811,E2 6557.811} C_VEL
LIN {X 0,Y 483.801,Z 1137.132,A -85,B 0,C 180,E1 6561.903,E2 6561.903} C_VEL
LIN {X 0,Y 483.59,Z 1143.442,A -85,B 0,C 180,E1 6566.409,E2 6566.409} C_VEL
LIN {X 0,Y 483.647,Z 1144.995,A -85,B 0,C 180,E1 6569.999,E2 6569.999} C_VEL
LIN {X 0,Y 483.624,Z 1143.357,A -85,B 0,C 180,E1 6573.589,E2 6573.589} C_VEL
LIN {X 0,Y 483.836,Z 1136.946,A -85,B 0,C 180,E1 6578.095,E2 6578.095} C_VEL
LIN {X 0,Y 484.296,Z 1125.248,A -85,B 0,C 180,E1 6582.641,E2 6582.641} C_VEL
LIN {X 0,Y 485.373,Z 1107.537,A -85,B 0,C 180,E1 6587.236,E2 6587.236} C_VEL
LIN {X 0,Y 487.33,Z 1085.062,A -85,B 0,C 180,E1 6591.462,E2 6591.462} C_VEL
LIN {X 0,Y 490.043,Z 1058.198,A -85,B 0,C 180,E1 6595.269,E2 6595.269} C_VEL
LIN {X 0,Y 493.24,Z 1027.472,A -85,B 0,C 180,E1 6598.582,E2 6598.582} C_VEL
LIN {X 0,Y 496.92,Z 991.895,A -85,B 0,C 180,E1 6601.455,E2 6601.455} C_VEL
LIN {X 0,Y 500.208,Z 955.957,A -85,B 0,C 180,E1 6603.588,E2 6603.588} C_VEL
LIN {X 0,Y 503.063,Z 916.937,A -85,B 0,C 180,E1 6605.098,E2 6605.098} C_VEL
LIN {X 0,Y 503.843,Z 885.45,A -85,B 0,C 180,E1 6605.871,E2 6605.871} C_VEL
LIN {X 0,Y 490.741,Z 858.924,A -85,B 0,C 180,E1 6607.679,E2 6607.679} C_VEL
LIN {X 0,Y 482.864,Z 845.004,A -85,B 0,C 180,E1 6608.805,E2 6608.805} C_VEL
LIN {X 0,Y 482.69,Z 843.44,A -85,B 0,C 180,E1 6608.856,E2 6608.856} C_VEL
LIN {X 0,Y 482.67,Z 843.44,A -85,B 0,C 180,E1 6613.83,E2 6613.83} C_VEL
LIN {X 0,Y 482.669,Z 843.44,A -85,B 0,C 180,E1 6618.839,E2 6618.839} C_VEL
LIN {X 0,Y 482.61,Z 843.44,A -85,B 0,C 180,E1 6624.657,E2 6624.657} C_VEL
LIN {X 0,Y 482.734,Z 843.44,A -85,B 0,C 180,E1 6629.883,E2 6629.883} C_VEL
LIN {X 0,Y 482.913,Z 843.44,A -85,B 0,C 180,E1 6635.95,E2 6635.95} C_VEL
LIN {X 0,Y 483.094,Z 843.44,A -85,B 0,C 180,E1 6641.738,E2 6641.738} C_VEL
LIN {X 0,Y 483.189,Z 843.44,A -85,B 0,C 180,E1 6647.331,E2 6647.331} C_VEL
LIN {X 0,Y 483.271,Z 843.44,A -85,B 0,C 180,E1 6652.802,E2 6652.802} C_VEL
LIN {X 0,Y 483.41,Z 843.44,A -85,B 0,C 180,E1 6658.206,E2 6658.206} C_VEL
LIN {X 0,Y 483.363,Z 843.44,A -85,B 0,C 180,E1 6663.592,E2 6663.592} C_VEL
LIN {X 0,Y 483.219,Z 843.44,A -85,B 0,C 180,E1 6669.013,E2 6669.013} C_VEL
LIN {X 0,Y 483.102,Z 843.44,A -85,B 0,C 180,E1 6674.52,E2 6674.52} C_VEL
LIN {X 0,Y 482.985,Z 843.44,A -85,B 0,C 180,E1 6680.171,E2 6680.171} C_VEL
LIN {X 0,Y 482.896,Z 843.44,A -85,B 0,C 180,E1 6686.036,E2 6686.036} C_VEL
LIN {X 0,Y 482.722,Z 843.44,A -85,B 0,C 180,E1 6692.22,E2 6692.22} C_VEL
LIN {X 0,Y 482.677,Z 843.44,A -85,B 0,C 180,E1 6698.853,E2 6698.853} C_VEL
LIN {X 0,Y 482.689,Z 843.44,A -85,B 0,C 180,E1 6703.824,E2 6703.824} C_VEL
LIN {X 0,Y 482.743,Z 843.44,A -85,B 0,C 180,E1 6706.306,E2 6706.306} C_VEL
LIN {X 0,Y 489.731,Z 858.126,A -85,B 0,C 180,E1 6707.276,E2 6707.276} C_VEL
LIN {X 0,Y 498.405,Z 874.201,A -85,B 0,C 180,E1 6708.339,E2 6708.339} C_VEL
LIN {X 0,Y 501.744,Z 883.746,A -85,B 0,C 180,E1 6708.804,E2 6708.804} C_VEL
LIN {X 0,Y 501.336,Z 908.272,A -85,B 0,C 180,E1 6709.366,E2 6709.366} C_VEL
LIN {X 0,Y 498.625,Z 951.61,A -85,B 0,C 180,E1 6710.85,E2 6710.85} C_VEL
LIN {X 0,Y 494.806,Z 993.701,A -85,B 0,C 180,E1 6713.066,E2 6713.066} C_VEL
LIN {X 0,Y 490.749,Z 1028.018,A -85,B 0,C 180,E1 6715.613,E2 6715.613} C_VEL
LIN {X 0,Y 486.41,Z 1062.208,A -85,B 0,C 180,E1 6718.988,E2 6718.988} C_VEL
LIN {X 0,Y 482.505,Z 1093.25,A -85,B 0,C 180,E1 6722.978,E2 6722.978} C_VEL
LIN {X 0,Y 479.402,Z 1120.379,A -85,B 0,C 180,E1 6727.526,E2 6727.526} C_VEL
LIN {X 0,Y 477.41,Z 1142.15,A -85,B 0,C 180,E1 6732.37,E2 6732.37} C_VEL
LIN {X 0,Y 476.304,Z 1157.769,A -85,B 0,C 180,E1 6737.144,E2 6737.144} C_VEL
LIN {X 0,Y 475.898,Z 1167.919,A -85,B 0,C 180,E1 6741.769,E2 6741.769} C_VEL
LIN {X 0,Y 475.699,Z 1173.628,A -85,B 0,C 180,E1 6746.351,E2 6746.351} C_VEL
LIN {X 0,Y 475.724,Z 1175,A -85,B 0,C 180,E1 6750.001,E2 6750.001} C_VEL
LIN {X 0,Y 475.686,Z 1173.627,A -85,B 0,C 180,E1 6753.651,E2 6753.651} C_VEL
LIN {X 0,Y 475.898,Z 1167.916,A -85,B 0,C 180,E1 6758.232,E2 6758.232} C_VEL
LIN {X 0,Y 476.227,Z 1157.766,A -85,B 0,C 180,E1 6762.86,E2 6762.86} C_VEL
LIN {X 0,Y 477.402,Z 1140.995,A -85,B 0,C 180,E1 6767.94,E2 6767.94} C_VEL
LIN {X 0,Y 479.558,Z 1118.319,A -85,B 0,C 180,E1 6772.879,E2 6772.879} C_VEL
LIN {X 0,Y 482.876,Z 1089.867,A -85,B 0,C 180,E1 6777.519,E2 6777.519} C_VEL
LIN {X 0,Y 487.178,Z 1056.732,A -85,B 0,C 180,E1 6781.617,E2 6781.617} C_VEL
LIN {X 0,Y 491.839,Z 1020.082,A -85,B 0,C 180,E1 6785.047,E2 6785.047} C_VEL
LIN {X 0,Y 495.773,Z 984.066,A -85,B 0,C 180,E1 6787.517,E2 6787.517} C_VEL
LIN {X 0,Y 499.36,Z 941.845,A -85,B 0,C 180,E1 6789.551,E2 6789.551} C_VEL
LIN {X 0,Y 501.776,Z 903.711,A -85,B 0,C 180,E1 6790.722,E2 6790.722} C_VEL
LIN {X 0,Y 501.516,Z 893.869,A -85,B 0,C 180,E1 6791.001,E2 6791.001} C_VEL
LIN {X 0,Y 474.769,Z 845.175,A -85,B 0,C 180,E1 6794.446,E2 6794.446} C_VEL
LIN {X 0,Y 474.554,Z 843.44,A -85,B 0,C 180,E1 6794.584,E2 6794.584} C_VEL
LIN {X 0,Y 474.687,Z 843.44,A -85,B 0,C 180,E1 6800.366,E2 6800.366} C_VEL
LIN {X 0,Y 474.829,Z 843.44,A -85,B 0,C 180,E1 6806.007,E2 6806.007} C_VEL
LIN {X 0,Y 474.921,Z 843.44,A -85,B 0,C 180,E1 6811.433,E2 6811.433} C_VEL
LIN {X 0,Y 474.907,Z 843.44,A -85,B 0,C 180,E1 6818.017,E2 6818.017} C_VEL
LIN {X 0,Y 482.547,Z 874.895,A -85,B 0,C 180,E1 6818.808,E2 6818.808} C_VEL
LIN {X 0,Y 482.136,Z 907.311,A -85,B 0,C 180,E1 6819.613,E2 6819.613} C_VEL
LIN {X 0,Y 481.195,Z 937.226,A -85,B 0,C 180,E1 6821.09,E2 6821.09} C_VEL
LIN {X 0,Y 479.896,Z 963.563,A -85,B 0,C 180,E1 6823.151,E2 6823.151} C_VEL
LIN {X 0,Y 478.486,Z 986.528,A -85,B 0,C 180,E1 6825.805,E2 6825.805} C_VEL
LIN {X 0,Y 477.409,Z 1005.401,A -85,B 0,C 180,E1 6829.031,E2 6829.031} C_VEL
LIN {X 0,Y 476.731,Z 1017.753,A -85,B 0,C 180,E1 6832.242,E2 6832.242} C_VEL
LIN {X 0,Y 476.413,Z 1025.256,A -85,B 0,C 180,E1 6835.442,E2 6835.442} C_VEL
LIN {X 0,Y 476.241,Z 1028.406,A -85,B 0,C 180,E1 6838.177,E2 6838.177} C_VEL
LIN {X 0,Y 476.239,Z 1028.194,A -85,B 0,C 180,E1 6841.821,E2 6841.821} C_VEL
LIN {X 0,Y 476.387,Z 1022.914,A -85,B 0,C 180,E1 6845.47,E2 6845.47} C_VEL
LIN {X 0,Y 476.824,Z 1012.03,A -85,B 0,C 180,E1 6849.134,E2 6849.134} C_VEL
LIN {X 0,Y 477.744,Z 995.379,A -85,B 0,C 180,E1 6852.583,E2 6852.583} C_VEL
LIN {X 0,Y 479.059,Z 974.037,A -85,B 0,C 180,E1 6855.551,E2 6855.551} C_VEL
LIN {X 0,Y 480.593,Z 948.25,A -85,B 0,C 180,E1 6858.005,E2 6858.005} C_VEL
LIN {X 0,Y 481.917,Z 919.558,A -85,B 0,C 180,E1 6859.813,E2 6859.813} C_VEL
LIN {X 0,Y 482.788,Z 887.56,A -85,B 0,C 180,E1 6860.991,E2 6860.991} C_VEL
LIN {X 0,Y 482.12,Z 868.446,A -85,B 0,C 180,E1 6861.391,E2 6861.391} C_VEL
LIN {X 0,Y 474.99,Z 843.44,A -85,B 0,C 180,E1 6862.134,E2 6862.134} C_VEL
LIN {X 0,Y 474.796,Z 843.44,A -85,B 0,C 180,E1 6868.573,E2 6868.573} C_VEL
LIN {X 0,Y 474.831,Z 843.44,A -85,B 0,C 180,E1 6875.022,E2 6875.022} C_VEL
LIN {X 0,Y 474.631,Z 843.44,A -85,B 0,C 180,E1 6880.036,E2 6880.036} C_VEL
LIN {X 0,Y 474.508,Z 843.44,A -85,B 0,C 180,E1 6885.41,E2 6885.41} C_VEL
LIN {X 0,Y 474.888,Z 844.183,A -85,B 0,C 180,E1 6890.209,E2 6890.209} C_VEL
LIN {X 0,Y 483.73,Z 860.004,A -85,B 0,C 180,E1 6891.482,E2 6891.482} C_VEL
LIN {X 0,Y 496.915,Z 885.482,A -85,B 0,C 180,E1 6893.354,E2 6893.354} C_VEL
LIN {X 0,Y 498.051,Z 892.745,A -85,B 0,C 180,E1 6893.626,E2 6893.626} C_VEL
LIN {X 0,Y 495.977,Z 932.36,A -85,B 0,C 180,E1 6894.736,E2 6894.736} C_VEL
LIN {X 0,Y 492.768,Z 969.728,A -85,B 0,C 180,E1 6896.486,E2 6896.486} C_VEL
LIN {X 0,Y 489.066,Z 1004.098,A -85,B 0,C 180,E1 6898.809,E2 6898.809} C_VEL
LIN {X 0,Y 484.999,Z 1037.671,A -85,B 0,C 180,E1 6901.883,E2 6901.883} C_VEL
LIN {X 0,Y 481.567,Z 1067.709,A -85,B 0,C 180,E1 6905.473,E2 6905.473} C_VEL
LIN {X 0,Y 478.823,Z 1094.003,A -85,B 0,C 180,E1 6909.644,E2 6909.644} C_VEL
LIN {X 0,Y 477.122,Z 1113.889,A -85,B 0,C 180,E1 6913.877,E2 6913.877} C_VEL
LIN {X 0,Y 476.173,Z 1129.583,A -85,B 0,C 180,E1 6918.536,E2 6918.536} C_VEL
LIN {X 0,Y 475.861,Z 1138.755,A -85,B 0,C 180,E1 6922.687,E2 6922.687} C_VEL
LIN {X 0,Y 475.686,Z 1143.441,A -85,B 0,C 180,E1 6926.349,E2 6926.349} C_VEL
LIN {X 0,Y 475.747,Z 1144.995,A -85,B 0,C 180,E1 6929.999,E2 6929.999} C_VEL
LIN {X 0,Y 475.721,Z 1143.358,A -85,B 0,C 180,E1 6933.649,E2 6933.649} C_VEL
LIN {X 0,Y 475.97,Z 1136.948,A -85,B 0,C 180,E1 6938.229,E2 6938.229} C_VEL
LIN {X 0,Y 476.475,Z 1125.249,A -85,B 0,C 180,E1 6942.852,E2 6942.852} C_VEL
LIN {X 0,Y 477.603,Z 1108.314,A -85,B 0,C 180,E1 6947.356,E2 6947.356} C_VEL
LIN {X 0,Y 479.759,Z 1085.063,A -85,B 0,C 180,E1 6951.819,E2 6951.819} C_VEL
LIN {X 0,Y 482.783,Z 1057.296,A -85,B 0,C 180,E1 6955.794,E2 6955.794} C_VEL
LIN {X 0,Y 486.423,Z 1025.75,A -85,B 0,C 180,E1 6959.214,E2 6959.214} C_VEL
LIN {X 0,Y 490.273,Z 993.102,A -85,B 0,C 180,E1 6961.932,E2 6961.932} C_VEL
LIN {X 0,Y 493.921,Z 956.297,A -85,B 0,C 180,E1 6964.15,E2 6964.15} C_VEL
LIN {X 0,Y 496.923,Z 918.255,A -85,B 0,C 180,E1 6965.646,E2 6965.646} C_VEL
LIN {X 0,Y 497.783,Z 888.18,A -85,B 0,C 180,E1 6966.409,E2 6966.409} C_VEL
LIN {X 0,Y 485.552,Z 863.377,A -85,B 0,C 180,E1 6968.159,E2 6968.159} C_VEL
LIN {X 0,Y 474.766,Z 844.395,A -85,B 0,C 180,E1 6969.71,E2 6969.71} C_VEL
LIN {X 0,Y 474.693,Z 843.44,A -85,B 0,C 180,E1 6969.934,E2 6969.934} C_VEL
LIN {X 0,Y 474.692,Z 843.44,A -85,B 0,C 180,E1 6975.442,E2 6975.442} C_VEL
LIN {X 0,Y 474.671,Z 843.44,A -85,B 0,C 180,E1 6980.366,E2 6980.366} C_VEL
LIN {X 0,Y 474.717,Z 843.44,A -85,B 0,C 180,E1 6987.171,E2 6987.171} C_VEL
LIN {X 0,Y 474.906,Z 843.44,A -85,B 0,C 180,E1 6993.494,E2 6993.494} C_VEL
LIN {X 0,Y 475.126,Z 843.44,A -85,B 0,C 180,E1 6999.483,E2 6999.483} C_VEL
LIN {X 0,Y 475.287,Z 843.44,A -85,B 0,C 180,E1 7005.238,E2 7005.238} C_VEL
LIN {X 0,Y 475.359,Z 843.44,A -85,B 0,C 180,E1 7011.215,E2 7011.215} C_VEL
LIN {X 0,Y 475.601,Z 843.44,A -85,B 0,C 180,E1 7016.351,E2 7016.351} C_VEL
LIN {X 0,Y 475.695,Z 843.44,A -85,B 0,C 180,E1 7021.825,E2 7021.825} C_VEL
LIN {X 0,Y 475.421,Z 843.44,A -85,B 0,C 180,E1 7027.319,E2 7027.319} C_VEL
LIN {X 0,Y 475.208,Z 843.44,A -85,B 0,C 180,E1 7032.887,E2 7032.887} C_VEL
LIN {X 0,Y 475.076,Z 843.44,A -85,B 0,C 180,E1 7038.584,E2 7038.584} C_VEL
LIN {X 0,Y 475.008,Z 843.44,A -85,B 0,C 180,E1 7044.478,E2 7044.478} C_VEL
LIN {X 0,Y 474.791,Z 843.44,A -85,B 0,C 180,E1 7050.677,E2 7050.677} C_VEL
LIN {X 0,Y 474.743,Z 843.44,A -85,B 0,C 180,E1 7057.295,E2 7057.295} C_VEL
LIN {X 0,Y 474.695,Z 843.44,A -85,B 0,C 180,E1 7062.81,E2 7062.81} C_VEL
LIN {X 0,Y 474.736,Z 843.581,A -85,B 0,C 180,E1 7065.518,E2 7065.518} C_VEL
LIN {X 0,Y 479.364,Z 853.378,A -85,B 0,C 180,E1 7066.194,E2 7066.194} C_VEL
LIN {X 0,Y 501.969,Z 895.73,A -85,B 0,C 180,E1 7069.077,E2 7069.077} C_VEL
LIN {X 0,Y 501.336,Z 908.272,A -85,B 0,C 180,E1 7069.366,E2 7069.366} C_VEL
LIN {X 0,Y 497.094,Z 925.287,A -85,B 0,C 180,E1 7069.564,E2 7069.564} C_VEL
LIN {X 0,Y 492.826,Z 940.908,A -85,B 0,C 180,E1 7069.873,E2 7069.873} C_VEL
LIN {X 0,Y 492.748,Z 941.923,A -85,B 0,C 180,E1 7069.916,E2 7069.916} C_VEL
LIN {X 0,Y 488.88,Z 984.889,A -85,B 0,C 180,E1 7072.023,E2 7072.023} C_VEL
LIN {X 0,Y 484.461,Z 1024.498,A -85,B 0,C 180,E1 7074.796,E2 7074.796} C_VEL
LIN {X 0,Y 479.844,Z 1059.385,A -85,B 0,C 180,E1 7078.159,E2 7078.159} C_VEL
LIN {X 0,Y 475.42,Z 1091.369,A -85,B 0,C 180,E1 7082.241,E2 7082.241} C_VEL
LIN {X 0,Y 471.858,Z 1119.576,A -85,B 0,C 180,E1 7086.981,E2 7086.981} C_VEL
LIN {X 0,Y 469.688,Z 1141.389,A -85,B 0,C 180,E1 7091.86,E2 7091.86} C_VEL
LIN {X 0,Y 468.453,Z 1157.769,A -85,B 0,C 180,E1 7096.924,E2 7096.924} C_VEL
LIN {X 0,Y 468.013,Z 1167.919,A -85,B 0,C 180,E1 7101.63,E2 7101.63} C_VEL
LIN {X 0,Y 467.812,Z 1173.628,A -85,B 0,C 180,E1 7106.289,E2 7106.289} C_VEL
LIN {X 0,Y 467.841,Z 1175,A -85,B 0,C 180,E1 7110.001,E2 7110.001} C_VEL
LIN {X 0,Y 467.798,Z 1173.627,A -85,B 0,C 180,E1 7113.712,E2 7113.712} C_VEL
LIN {X 0,Y 468.01,Z 1167.916,A -85,B 0,C 180,E1 7118.372,E2 7118.372} C_VEL
LIN {X 0,Y 468.372,Z 1157.765,A -85,B 0,C 180,E1 7123.08,E2 7123.08} C_VEL
LIN {X 0,Y 469.609,Z 1141.593,A -85,B 0,C 180,E1 7128.086,E2 7128.086} C_VEL
LIN {X 0,Y 471.867,Z 1119.541,A -85,B 0,C 180,E1 7133.025,E2 7133.025} C_VEL
LIN {X 0,Y 475.347,Z 1091.836,A -85,B 0,C 180,E1 7137.689,E2 7137.689} C_VEL
LIN {X 0,Y 480.045,Z 1058.187,A -85,B 0,C 180,E1 7141.974,E2 7141.974} C_VEL
LIN {X 0,Y 484.467,Z 1024.548,A -85,B 0,C 180,E1 7145.199,E2 7145.199} C_VEL
LIN {X 0,Y 488.813,Z 986.174,A -85,B 0,C 180,E1 7147.893,E2 7147.893} C_VEL
LIN {X 0,Y 492.416,Z 947.583,A -85,B 0,C 180,E1 7149.84,E2 7149.84} C_VEL
LIN {X 0,Y 495.136,Z 908.964,A -85,B 0,C 180,E1 7151.14,E2 7151.14} C_VEL
LIN {X 0,Y 495.231,Z 897.15,A -85,B 0,C 180,E1 7151.46,E2 7151.46} C_VEL
LIN {X 0,Y 466.72,Z 844.544,A -85,B 0,C 180,E1 7155.339,E2 7155.339} C_VEL
LIN {X 0,Y 466.632,Z 843.44,A -85,B 0,C 180,E1 7155.551,E2 7155.551} C_VEL
LIN {X 0,Y 466.785,Z 843.44,A -85,B 0,C 180,E1 7161.957,E2 7161.957} C_VEL
LIN {X 0,Y 466.934,Z 843.44,A -85,B 0,C 180,E1 7168.749,E2 7168.749} C_VEL
LIN {X 0,Y 466.987,Z 843.44,A -85,B 0,C 180,E1 7175.213,E2 7175.213} C_VEL
LIN {X 0,Y 467.011,Z 843.44,A -85,B 0,C 180,E1 7177.681,E2 7177.681} C_VEL
LIN {X 0,Y 474.981,Z 875.093,A -85,B 0,C 180,E1 7178.529,E2 7178.529} C_VEL
LIN {X 0,Y 474.655,Z 907.569,A -85,B 0,C 180,E1 7179.317,E2 7179.317} C_VEL
LIN {X 0,Y 473.73,Z 937.425,A -85,B 0,C 180,E1 7180.772,E2 7180.772} C_VEL
LIN {X 0,Y 472.392,Z 964.402,A -85,B 0,C 180,E1 7182.875,E2 7182.875} C_VEL
LIN {X 0,Y 470.909,Z 987.647,A -85,B 0,C 180,E1 7185.571,E2 7185.571} C_VEL
LIN {X 0,Y 469.839,Z 1005.56,A -85,B 0,C 180,E1 7188.616,E2 7188.616} C_VEL
LIN {X 0,Y 469.024,Z 1019.149,A -85,B 0,C 180,E1 7192.114,E2 7192.114} C_VEL
LIN {X 0,Y 468.673,Z 1026.689,A -85,B 0,C 180,E1 7195.367,E2 7195.367} C_VEL
LIN {X 0,Y 468.475,Z 1029.834,A -85,B 0,C 180,E1 7198.147,E2 7198.147} C_VEL
LIN {X 0,Y 468.472,Z 1029.568,A -85,B 0,C 180,E1 7201.851,E2 7201.851} C_VEL
LIN {X 0,Y 468.641,Z 1024.199,A -85,B 0,C 180,E1 7205.561,E2 7205.561} C_VEL
LIN {X 0,Y 469.1,Z 1013.192,A -85,B 0,C 180,E1 7209.285,E2 7209.285} C_VEL
LIN {X 0,Y 470.104,Z 996.356,A -85,B 0,C 180,E1 7212.791,E2 7212.791} C_VEL
LIN {X 0,Y 471.449,Z 975.139,A -85,B 0,C 180,E1 7215.768,E2 7215.768} C_VEL
LIN {X 0,Y 472.997,Z 950.213,A -85,B 0,C 180,E1 7218.183,E2 7218.183} C_VEL
LIN {X 0,Y 474.365,Z 922.174,A -85,B 0,C 180,E1 7220.006,E2 7220.006} C_VEL
LIN {X 0,Y 475.272,Z 890.807,A -85,B 0,C 180,E1 7221.222,E2 7221.222} C_VEL
LIN {X 0,Y 474.58,Z 869.791,A -85,B 0,C 180,E1 7221.684,E2 7221.684} C_VEL
LIN {X 0,Y 467.053,Z 843.44,A -85,B 0,C 180,E1 7222.464,E2 7222.464} C_VEL
LIN {X 0,Y 466.864,Z 843.44,A -85,B 0,C 180,E1 7229.104,E2 7229.104} C_VEL
LIN {X 0,Y 466.887,Z 843.44,A -85,B 0,C 180,E1 7233.452,E2 7233.452} C_VEL
LIN {X 0,Y 466.68,Z 843.44,A -85,B 0,C 180,E1 7240.451,E2 7240.451} C_VEL
LIN {X 0,Y 466.625,Z 843.44,A -85,B 0,C 180,E1 7247.044,E2 7247.044} C_VEL
LIN {X 0,Y 466.783,Z 843.44,A -85,B 0,C 180,E1 7249.247,E2 7249.247} C_VEL
LIN {X 0,Y 469.151,Z 849.028,A -85,B 0,C 180,E1 7249.652,E2 7249.652} C_VEL
LIN {X 0,Y 488.983,Z 883.833,A -85,B 0,C 180,E1 7252.501,E2 7252.501} C_VEL
LIN {X 0,Y 492.115,Z 891.23,A -85,B 0,C 180,E1 7252.99,E2 7252.99} C_VEL
LIN {X 0,Y 490.091,Z 930.157,A -85,B 0,C 180,E1 7254.054,E2 7254.054} C_VEL
LIN {X 0,Y 486.719,Z 967.98,A -85,B 0,C 180,E1 7255.795,E2 7255.795} C_VEL
LIN {X 0,Y 482.799,Z 1001.962,A -85,B 0,C 180,E1 7258.07,E2 7258.07} C_VEL
LIN {X 0,Y 478.505,Z 1034.271,A -85,B 0,C 180,E1 7260.997,E2 7260.997} C_VEL
LIN {X 0,Y 474.298,Z 1067.035,A -85,B 0,C 180,E1 7264.976,E2 7264.976} C_VEL
LIN {X 0,Y 471.377,Z 1092.006,A -85,B 0,C 180,E1 7268.938,E2 7268.938} C_VEL
LIN {X 0,Y 469.538,Z 1111.934,A -85,B 0,C 180,E1 7273.128,E2 7273.128} C_VEL
LIN {X 0,Y 468.428,Z 1126.903,A -85,B 0,C 180,E1 7277.397,E2 7277.397} C_VEL
LIN {X 0,Y 468.042,Z 1137.129,A -85,B 0,C 180,E1 7281.628,E2 7281.628} C_VEL
LIN {X 0,Y 467.797,Z 1143.441,A -85,B 0,C 180,E1 7286.288,E2 7286.288} C_VEL
LIN {X 0,Y 467.858,Z 1144.995,A -85,B 0,C 180,E1 7289.999,E2 7289.999} C_VEL
LIN {X 0,Y 467.83,Z 1143.359,A -85,B 0,C 180,E1 7293.71,E2 7293.71} C_VEL
LIN {X 0,Y 468.086,Z 1136.949,A -85,B 0,C 180,E1 7298.369,E2 7298.369} C_VEL
LIN {X 0,Y 468.65,Z 1125.251,A -85,B 0,C 180,E1 7303.07,E2 7303.07} C_VEL
LIN {X 0,Y 470.007,Z 1107.055,A -85,B 0,C 180,E1 7307.927,E2 7307.927} C_VEL
LIN {X 0,Y 472.239,Z 1084.464,A -85,B 0,C 180,E1 7312.287,E2 7312.287} C_VEL
LIN {X 0,Y 475.455,Z 1057.3,A -85,B 0,C 180,E1 7316.222,E2 7316.222} C_VEL
LIN {X 0,Y 479.552,Z 1026.694,A -85,B 0,C 180,E1 7319.674,E2 7319.674} C_VEL
LIN {X 0,Y 483.884,Z 992.917,A -85,B 0,C 180,E1 7322.52,E2 7322.52} C_VEL
LIN {X 0,Y 487.75,Z 956.499,A -85,B 0,C 180,E1 7324.736,E2 7324.736} C_VEL
LIN {X 0,Y 490.952,Z 917.433,A -85,B 0,C 180,E1 7326.276,E2 7326.276} C_VEL
LIN {X 0,Y 491.896,Z 891.244,A -85,B 0,C 180,E1 7326.942,E2 7326.942} C_VEL
LIN {X 0,Y 479.111,Z 865.495,A -85,B 0,C 180,E1 7328.831,E2 7328.831} C_VEL
LIN {X 0,Y 466.83,Z 844.755,A -85,B 0,C 180,E1 7330.607,E2 7330.607} C_VEL
LIN {X 0,Y 466.725,Z 843.44,A -85,B 0,C 180,E1 7330.824,E2 7330.824} C_VEL
LIN {X 0,Y 466.799,Z 843.44,A -85,B 0,C 180,E1 7337.073,E2 7337.073} C_VEL
LIN {X 0,Y 466.716,Z 843.44,A -85,B 0,C 180,E1 7341.953,E2 7341.953} C_VEL
LIN {X 0,Y 466.802,Z 843.44,A -85,B 0,C 180,E1 7348.742,E2 7348.742} C_VEL
LIN {X 0,Y 467.068,Z 843.44,A -85,B 0,C 180,E1 7355.187,E2 7355.187} C_VEL
LIN {X 0,Y 467.22,Z 843.44,A -85,B 0,C 180,E1 7361.094,E2 7361.094} C_VEL
LIN {X 0,Y 467.356,Z 843.44,A -85,B 0,C 180,E1 7366.895,E2 7366.895} C_VEL
LIN {X 0,Y 467.448,Z 843.44,A -85,B 0,C 180,E1 7372.557,E2 7372.557} C_VEL
LIN {X 0,Y 467.638,Z 843.44,A -85,B 0,C 180,E1 7378.146,E2 7378.146} C_VEL
LIN {X 0,Y 467.549,Z 843.44,A -85,B 0,C 180,E1 7383.714,E2 7383.714} C_VEL
LIN {X 0,Y 467.393,Z 843.44,A -85,B 0,C 180,E1 7389.321,E2 7389.321} C_VEL
LIN {X 0,Y 467.23,Z 843.44,A -85,B 0,C 180,E1 7395.025,E2 7395.025} C_VEL
LIN {X 0,Y 467.115,Z 843.44,A -85,B 0,C 180,E1 7400.887,E2 7400.887} C_VEL
LIN {X 0,Y 466.97,Z 843.44,A -85,B 0,C 180,E1 7406.994,E2 7406.994} C_VEL
LIN {X 0,Y 466.798,Z 843.44,A -85,B 0,C 180,E1 7413.461,E2 7413.461} C_VEL
LIN {X 0,Y 466.75,Z 843.44,A -85,B 0,C 180,E1 7420.446,E2 7420.446} C_VEL
LIN {X 0,Y 466.814,Z 843.44,A -85,B 0,C 180,E1 7424.615,E2 7424.615} C_VEL
LIN {X 0,Y 471.544,Z 853.529,A -85,B 0,C 180,E1 7425.384,E2 7425.384} C_VEL
LIN {X 0,Y 495.475,Z 897.973,A -85,B 0,C 180,E1 7428.584,E2 7428.584} C_VEL
LIN {X 0,Y 492.748,Z 941.923,A -85,B 0,C 180,E1 7429.916,E2 7429.916} C_VEL
LIN {X 0,Y 488.332,Z 958.558,A -85,B 0,C 180,E1 7430.388,E2 7430.388} C_VEL
LIN {X 0,Y 483.381,Z 974.608,A -85,B 0,C 180,E1 7430.927,E2 7430.927} C_VEL
LIN {X 0,Y 479.104,Z 1012.589,A -85,B 0,C 180,E1 7433.382,E2 7433.382} C_VEL
LIN {X 0,Y 474.385,Z 1048.625,A -85,B 0,C 180,E1 7436.511,E2 7436.511} C_VEL
LIN {X 0,Y 469.605,Z 1081.127,A -85,B 0,C 180,E1 7440.318,E2 7440.318} C_VEL
LIN {X 0,Y 465.413,Z 1111.044,A -85,B 0,C 180,E1 7444.981,E2 7444.981} C_VEL
LIN {X 0,Y 462.431,Z 1134.852,A -85,B 0,C 180,E1 7449.892,E2 7449.892} C_VEL
LIN {X 0,Y 460.94,Z 1152.295,A -85,B 0,C 180,E1 7454.765,E2 7454.765} C_VEL
LIN {X 0,Y 460.228,Z 1164.406,A -85,B 0,C 180,E1 7459.576,E2 7459.576} C_VEL
LIN {X 0,Y 460.012,Z 1171.905,A -85,B 0,C 180,E1 7464.334,E2 7464.334} C_VEL
LIN {X 0,Y 460.007,Z 1174.657,A -85,B 0,C 180,E1 7468.115,E2 7468.115} C_VEL
LIN {X 0,Y 459.871,Z 1174.657,A -85,B 0,C 180,E1 7471.888,E2 7471.888} C_VEL
LIN {X 0,Y 460.028,Z 1170.702,A -85,B 0,C 180,E1 7476.616,E2 7476.616} C_VEL
LIN {X 0,Y 460.322,Z 1162.432,A -85,B 0,C 180,E1 7481.383,E2 7481.383} C_VEL
LIN {X 0,Y 461.308,Z 1147.678,A -85,B 0,C 180,E1 7486.691,E2 7486.691} C_VEL
LIN {X 0,Y 463.373,Z 1127.372,A -85,B 0,C 180,E1 7491.806,E2 7491.806} C_VEL
LIN {X 0,Y 466.752,Z 1101.025,A -85,B 0,C 180,E1 7496.734,E2 7496.734} C_VEL
LIN {X 0,Y 471.416,Z 1069.63,A -85,B 0,C 180,E1 7501.159,E2 7501.159} C_VEL
LIN {X 0,Y 475.833,Z 1037.86,A -85,B 0,C 180,E1 7504.516,E2 7504.516} C_VEL
LIN {X 0,Y 480.46,Z 1000.901,A -85,B 0,C 180,E1 7507.459,E2 7507.459} C_VEL
LIN {X 0,Y 484.692,Z 961.83,A -85,B 0,C 180,E1 7509.729,E2 7509.729} C_VEL
LIN {X 0,Y 487.835,Z 921.352,A -85,B 0,C 180,E1 7511.342,E2 7511.342} C_VEL
LIN {X 0,Y 488.63,Z 899.809,A -85,B 0,C 180,E1 7511.96,E2 7511.96} C_VEL
LIN {X 0,Y 460.543,Z 848.498,A -85,B 0,C 180,E1 7515.961,E2 7515.961} C_VEL
LIN {X 0,Y 458.702,Z 843.44,A -85,B 0,C 180,E1 7516.378,E2 7516.378} C_VEL
LIN {X 0,Y 458.866,Z 843.44,A -85,B 0,C 180,E1 7522.368,E2 7522.368} C_VEL
LIN {X 0,Y 459.026,Z 843.44,A -85,B 0,C 180,E1 7529.053,E2 7529.053} C_VEL
LIN {X 0,Y 459.029,Z 843.44,A -85,B 0,C 180,E1 7534.61,E2 7534.61} C_VEL
LIN {X 0,Y 459.08,Z 843.44,A -85,B 0,C 180,E1 7537.349,E2 7537.349} C_VEL
LIN {X 0,Y 467.473,Z 876.155,A -85,B 0,C 180,E1 7538.251,E2 7538.251} C_VEL
LIN {X 0,Y 467.153,Z 909.41,A -85,B 0,C 180,E1 7539.066,E2 7539.066} C_VEL
LIN {X 0,Y 466.148,Z 939.718,A -85,B 0,C 180,E1 7540.574,E2 7540.574} C_VEL
LIN {X 0,Y 464.817,Z 966.472,A -85,B 0,C 180,E1 7542.709,E2 7542.709} C_VEL
LIN {X 0,Y 463.335,Z 988.794,A -85,B 0,C 180,E1 7545.33,E2 7545.33} C_VEL
LIN {X 0,Y 462.202,Z 1006.864,A -85,B 0,C 180,E1 7548.426,E2 7548.426} C_VEL
LIN {X 0,Y 461.315,Z 1020.544,A -85,B 0,C 180,E1 7551.982,E2 7551.982} C_VEL
LIN {X 0,Y 460.951,Z 1028.119,A -85,B 0,C 180,E1 7555.289,E2 7555.289} C_VEL
LIN {X 0,Y 460.716,Z 1031.26,A -85,B 0,C 180,E1 7558.116,E2 7558.116} C_VEL
LIN {X 0,Y 460.713,Z 1030.941,A -85,B 0,C 180,E1 7561.882,E2 7561.882} C_VEL
LIN {X 0,Y 460.894,Z 1025.484,A -85,B 0,C 180,E1 7565.654,E2 7565.654} C_VEL
LIN {X 0,Y 461.401,Z 1014.344,A -85,B 0,C 180,E1 7569.442,E2 7569.442} C_VEL
LIN {X 0,Y 462.451,Z 997.331,A -85,B 0,C 180,E1 7573.006,E2 7573.006} C_VEL
LIN {X 0,Y 463.877,Z 975.917,A -85,B 0,C 180,E1 7576.031,E2 7576.031} C_VEL
LIN {X 0,Y 465.499,Z 950.684,A -85,B 0,C 180,E1 7578.487,E2 7578.487} C_VEL
LIN {X 0,Y 466.915,Z 922.099,A -85,B 0,C 180,E1 7580.343,E2 7580.343} C_VEL
LIN {X 0,Y 467.842,Z 890.066,A -85,B 0,C 180,E1 7581.566,E2 7581.566} C_VEL
LIN {X 0,Y 467.169,Z 871.426,A -85,B 0,C 180,E1 7581.976,E2 7581.976} C_VEL
LIN {X 0,Y 459.106,Z 843.44,A -85,B 0,C 180,E1 7582.9,E2 7582.9} C_VEL
LIN {X 0,Y 458.901,Z 843.44,A -85,B 0,C 180,E1 7589.659,E2 7589.659} C_VEL
LIN {X 0,Y 458.859,Z 843.44,A -85,B 0,C 180,E1 7596.432,E2 7596.432} C_VEL
LIN {X 0,Y 458.721,Z 843.44,A -85,B 0,C 180,E1 7601.304,E2 7601.304} C_VEL
LIN {X 0,Y 458.779,Z 843.44,A -85,B 0,C 180,E1 7608.304,E2 7608.304} C_VEL
LIN {X 0,Y 461.297,Z 849.181,A -85,B 0,C 180,E1 7608.735,E2 7608.735} C_VEL
LIN {X 0,Y 483.47,Z 887.481,A -85,B 0,C 180,E1 7611.981,E2 7611.981} C_VEL
LIN {X 0,Y 486.176,Z 895.366,A -85,B 0,C 180,E1 7612.453,E2 7612.453} C_VEL
LIN {X 0,Y 483.7,Z 935.461,A -85,B 0,C 180,E1 7613.629,E2 7613.629} C_VEL
LIN {X 0,Y 479.829,Z 973.985,A -85,B 0,C 180,E1 7615.525,E2 7615.525} C_VEL
LIN {X 0,Y 475.142,Z 1010.803,A -85,B 0,C 180,E1 7618.191,E2 7618.191} C_VEL
LIN {X 0,Y 470.405,Z 1043.628,A -85,B 0,C 180,E1 7621.471,E2 7621.471} C_VEL
LIN {X 0,Y 466.098,Z 1073.252,A -85,B 0,C 180,E1 7625.43,E2 7625.43} C_VEL
LIN {X 0,Y 463.07,Z 1098.906,A -85,B 0,C 180,E1 7629.919,E2 7629.919} C_VEL
LIN {X 0,Y 461.306,Z 1117.488,A -85,B 0,C 180,E1 7634.288,E2 7634.288} C_VEL
LIN {X 0,Y 460.391,Z 1131.965,A -85,B 0,C 180,E1 7639.099,E2 7639.099} C_VEL
LIN {X 0,Y 460.044,Z 1140.283,A -85,B 0,C 180,E1 7643.384,E2 7643.384} C_VEL
LIN {X 0,Y 459.882,Z 1144.61,A -85,B 0,C 180,E1 7648.112,E2 7648.112} C_VEL
LIN {X 0,Y 460,Z 1144.56,A -85,B 0,C 180,E1 7651.885,E2 7651.885} C_VEL
LIN {X 0,Y 460.019,Z 1140.161,A -85,B 0,C 180,E1 7656.614,E2 7656.614} C_VEL
LIN {X 0,Y 460.439,Z 1130.606,A -85,B 0,C 180,E1 7661.379,E2 7661.379} C_VEL
LIN {X 0,Y 461.521,Z 1115.435,A -85,B 0,C 180,E1 7666.191,E2 7666.191} C_VEL
LIN {X 0,Y 463.671,Z 1093.522,A -85,B 0,C 180,E1 7671.051,E2 7671.051} C_VEL
LIN {X 0,Y 467.328,Z 1065.104,A -85,B 0,C 180,E1 7675.679,E2 7675.679} C_VEL
LIN {X 0,Y 471.524,Z 1035.587,A -85,B 0,C 180,E1 7679.33,E2 7679.33} C_VEL
LIN {X 0,Y 476.306,Z 1001.696,A -85,B 0,C 180,E1 7682.466,E2 7682.466} C_VEL
LIN {X 0,Y 480.943,Z 963.756,A -85,B 0,C 180,E1 7684.975,E2 7684.975} C_VEL
LIN {X 0,Y 484.691,Z 923.417,A -85,B 0,C 180,E1 7686.709,E2 7686.709} C_VEL
LIN {X 0,Y 485.881,Z 893.751,A -85,B 0,C 180,E1 7687.523,E2 7687.523} C_VEL
LIN {X 0,Y 473.603,Z 869.635,A -85,B 0,C 180,E1 7689.36,E2 7689.36} C_VEL
LIN {X 0,Y 458.905,Z 844.307,A -85,B 0,C 180,E1 7691.558,E2 7691.558} C_VEL
LIN {X 0,Y 458.857,Z 843.44,A -85,B 0,C 180,E1 7691.86,E2 7691.86} C_VEL
LIN {X 0,Y 458.857,Z 843.44,A -85,B 0,C 180,E1 7698.711,E2 7698.711} C_VEL
LIN {X 0,Y 458.789,Z 843.44,A -85,B 0,C 180,E1 7705.594,E2 7705.594} C_VEL
LIN {X 0,Y 458.885,Z 843.44,A -85,B 0,C 180,E1 7710.339,E2 7710.339} C_VEL
LIN {X 0,Y 459.141,Z 843.44,A -85,B 0,C 180,E1 7716.693,E2 7716.693} C_VEL
LIN {X 0,Y 459.412,Z 843.44,A -85,B 0,C 180,E1 7722.895,E2 7722.895} C_VEL
LIN {X 0,Y 459.46,Z 843.44,A -85,B 0,C 180,E1 7728.598,E2 7728.598} C_VEL
LIN {X 0,Y 459.604,Z 843.44,A -85,B 0,C 180,E1 7734.33,E2 7734.33} C_VEL
LIN {X 0,Y 459.834,Z 843.44,A -85,B 0,C 180,E1 7740.001,E2 7740.001} C_VEL
LIN {X 0,Y 459.644,Z 843.44,A -85,B 0,C 180,E1 7745.672,E2 7745.672} C_VEL
LIN {X 0,Y 459.419,Z 843.44,A -85,B 0,C 180,E1 7751.405,E2 7751.405} C_VEL
LIN {X 0,Y 459.252,Z 843.44,A -85,B 0,C 180,E1 7757.26,E2 7757.26} C_VEL
LIN {X 0,Y 459.141,Z 843.44,A -85,B 0,C 180,E1 7763.309,E2 7763.309} C_VEL
LIN {X 0,Y 458.892,Z 843.44,A -85,B 0,C 180,E1 7769.662,E2 7769.662} C_VEL
LIN {X 0,Y 458.805,Z 843.44,A -85,B 0,C 180,E1 7776.439,E2 7776.439} C_VEL
LIN {X 0,Y 458.87,Z 843.44,A -85,B 0,C 180,E1 7781.29,E2 7781.29} C_VEL
LIN {X 0,Y 458.876,Z 843.806,A -85,B 0,C 180,E1 7783.74,E2 7783.74} C_VEL
LIN {X 0,Y 461.541,Z 849.353,A -85,B 0,C 180,E1 7784.176,E2 7784.176} C_VEL
LIN {X 0,Y 488.982,Z 901.89,A -85,B 0,C 180,E1 7788.132,E2 7788.132} C_VEL
LIN {X 0,Y 486.112,Z 943.808,A -85,B 0,C 180,E1 7789.457,E2 7789.457} C_VEL
LIN {X 0,Y 483.381,Z 974.608,A -85,B 0,C 180,E1 7790.927,E2 7790.927} C_VEL
LIN {X 0,Y 477.992,Z 990.619,A -85,B 0,C 180,E1 7791.579,E2 7791.579} C_VEL
LIN {X 0,Y 473.216,Z 1004.921,A -85,B 0,C 180,E1 7792.301,E2 7792.301} C_VEL
LIN {X 0,Y 473.142,Z 1005.835,A -85,B 0,C 180,E1 7792.369,E2 7792.369} C_VEL
LIN {X 0,Y 468.225,Z 1041.729,A -85,B 0,C 180,E1 7795.366,E2 7795.366} C_VEL
LIN {X 0,Y 463.415,Z 1075.012,A -85,B 0,C 180,E1 7799.03,E2 7799.03} C_VEL
LIN {X 0,Y 459.007,Z 1103.692,A -85,B 0,C 180,E1 7803.262,E2 7803.262} C_VEL
LIN {X 0,Y 455.669,Z 1128.41,A -85,B 0,C 180,E1 7808.049,E2 7808.049} C_VEL
LIN {X 0,Y 453.619,Z 1147.686,A -85,B 0,C 180,E1 7813.019,E2 7813.019} C_VEL
LIN {X 0,Y 452.416,Z 1162.435,A -85,B 0,C 180,E1 7818.417,E2 7818.417} C_VEL
LIN {X 0,Y 452.128,Z 1170.703,A -85,B 0,C 180,E1 7823.27,E2 7823.27} C_VEL
LIN {X 0,Y 452.099,Z 1174.657,A -85,B 0,C 180,E1 7828.082,E2 7828.082} C_VEL
LIN {X 0,Y 451.979,Z 1174.657,A -85,B 0,C 180,E1 7831.921,E2 7831.921} C_VEL
LIN {X 0,Y 452.137,Z 1170.702,A -85,B 0,C 180,E1 7836.732,E2 7836.732} C_VEL
LIN {X 0,Y 452.445,Z 1162.431,A -85,B 0,C 180,E1 7841.584,E2 7841.584} C_VEL
LIN {X 0,Y 453.54,Z 1147.679,A -85,B 0,C 180,E1 7846.986,E2 7846.986} C_VEL
LIN {X 0,Y 455.932,Z 1126.169,A -85,B 0,C 180,E1 7852.453,E2 7852.453} C_VEL
LIN {X 0,Y 459.66,Z 1099.356,A -85,B 0,C 180,E1 7857.463,E2 7857.463} C_VEL
LIN {X 0,Y 464.064,Z 1071.009,A -85,B 0,C 180,E1 7861.47,E2 7861.47} C_VEL
LIN {X 0,Y 469.174,Z 1035.476,A -85,B 0,C 180,E1 7865.223,E2 7865.223} C_VEL
LIN {X 0,Y 474.265,Z 996.687,A -85,B 0,C 180,E1 7868.271,E2 7868.271} C_VEL
LIN {X 0,Y 478.81,Z 955.114,A -85,B 0,C 180,E1 7870.588,E2 7870.588} C_VEL
LIN {X 0,Y 481.947,Z 915.289,A -85,B 0,C 180,E1 7872.073,E2 7872.073} C_VEL
LIN {X 0,Y 482.047,Z 902.655,A -85,B 0,C 180,E1 7872.469,E2 7872.469} C_VEL
LIN {X 0,Y 455.992,Z 854.084,A -85,B 0,C 180,E1 7876.377,E2 7876.377} C_VEL
LIN {X 0,Y 450.915,Z 844.872,A -85,B 0,C 180,E1 7877.21,E2 7877.21} C_VEL
LIN {X 0,Y 450.771,Z 843.44,A -85,B 0,C 180,E1 7877.324,E2 7877.324} C_VEL
LIN {X 0,Y 451.003,Z 843.44,A -85,B 0,C 180,E1 7883.683,E2 7883.683} C_VEL
LIN {X 0,Y 451.085,Z 843.44,A -85,B 0,C 180,E1 7889.772,E2 7889.772} C_VEL
LIN {X 0,Y 451.129,Z 843.44,A -85,B 0,C 180,E1 7896.662,E2 7896.662} C_VEL
LIN {X 0,Y 451.209,Z 844.313,A -85,B 0,C 180,E1 7896.997,E2 7896.997} C_VEL
LIN {X 0,Y 460.018,Z 879.121,A -85,B 0,C 180,E1 7897.991,E2 7897.991} C_VEL
LIN {X 0,Y 459.64,Z 912.093,A -85,B 0,C 180,E1 7898.837,E2 7898.837} C_VEL
LIN {X 0,Y 458.656,Z 941.93,A -85,B 0,C 180,E1 7900.364,E2 7900.364} C_VEL
LIN {X 0,Y 457.232,Z 968.623,A -85,B 0,C 180,E1 7902.537,E2 7902.537} C_VEL
LIN {X 0,Y 455.69,Z 991.627,A -85,B 0,C 180,E1 7905.325,E2 7905.325} C_VEL
LIN {X 0,Y 454.467,Z 1009.327,A -85,B 0,C 180,E1 7908.469,E2 7908.469} C_VEL
LIN {X 0,Y 453.613,Z 1021.952,A -85,B 0,C 180,E1 7911.845,E2 7911.845} C_VEL
LIN {X 0,Y 453.227,Z 1029.553,A -85,B 0,C 180,E1 7915.209,E2 7915.209} C_VEL
LIN {X 0,Y 452.963,Z 1032.685,A -85,B 0,C 180,E1 7918.084,E2 7918.084} C_VEL
LIN {X 0,Y 452.96,Z 1032.312,A -85,B 0,C 180,E1 7921.914,E2 7921.914} C_VEL
LIN {X 0,Y 453.161,Z 1026.765,A -85,B 0,C 180,E1 7925.751,E2 7925.751} C_VEL
LIN {X 0,Y 453.693,Z 1015.493,A -85,B 0,C 180,E1 7929.604,E2 7929.604} C_VEL
LIN {X 0,Y 454.807,Z 998.306,A -85,B 0,C 180,E1 7933.229,E2 7933.229} C_VEL
LIN {X 0,Y 456.308,Z 976.857,A -85,B 0,C 180,E1 7936.28,E2 7936.28} C_VEL
LIN {X 0,Y 457.999,Z 951.11,A -85,B 0,C 180,E1 7938.801,E2 7938.801} C_VEL
LIN {X 0,Y 459.496,Z 921.618,A -85,B 0,C 180,E1 7940.708,E2 7940.708} C_VEL
LIN {X 0,Y 460.4,Z 890.515,A -85,B 0,C 180,E1 7941.885,E2 7941.885} C_VEL
LIN {X 0,Y 459.698,Z 873.04,A -85,B 0,C 180,E1 7942.279,E2 7942.279} C_VEL
LIN {X 0,Y 451.171,Z 843.44,A -85,B 0,C 180,E1 7943.297,E2 7943.297} C_VEL
LIN {X 0,Y 450.996,Z 843.44,A -85,B 0,C 180,E1 7950.233,E2 7950.233} C_VEL
LIN {X 0,Y 450.94,Z 843.44,A -85,B 0,C 180,E1 7957.178,E2 7957.178} C_VEL
LIN {X 0,Y 450.725,Z 843.44,A -85,B 0,C 180,E1 7962.348,E2 7962.348} C_VEL
LIN {X 0,Y 450.831,Z 843.997,A -85,B 0,C 180,E1 7967.335,E2 7967.335} C_VEL
LIN {X 0,Y 453.382,Z 849.254,A -85,B 0,C 180,E1 7967.766,E2 7967.766} C_VEL
LIN {X 0,Y 477.906,Z 891.103,A -85,B 0,C 180,E1 7971.449,E2 7971.449} C_VEL
LIN {X 0,Y 480.292,Z 897.737,A -85,B 0,C 180,E1 7971.863,E2 7971.863} C_VEL
LIN {X 0,Y 477.38,Z 939.466,A -85,B 0,C 180,E1 7973.145,E2 7973.145} C_VEL
LIN {X 0,Y 473.272,Z 977.529,A -85,B 0,C 180,E1 7975.118,E2 7975.118} C_VEL
LIN {X 0,Y 468.282,Z 1013.356,A -85,B 0,C 180,E1 7977.814,E2 7977.814} C_VEL
LIN {X 0,Y 463.269,Z 1045.607,A -85,B 0,C 180,E1 7981.138,E2 7981.138} C_VEL
LIN {X 0,Y 458.826,Z 1073.899,A -85,B 0,C 180,E1 7985.015,E2 7985.015} C_VEL
LIN {X 0,Y 455.435,Z 1098.9,A -85,B 0,C 180,E1 7989.568,E2 7989.568} C_VEL
LIN {X 0,Y 453.524,Z 1117.485,A -85,B 0,C 180,E1 7994.011,E2 7994.011} C_VEL
LIN {X 0,Y 452.537,Z 1131.963,A -85,B 0,C 180,E1 7998.907,E2 7998.907} C_VEL
LIN {X 0,Y 452.152,Z 1140.281,A -85,B 0,C 180,E1 8003.268,E2 8003.268} C_VEL
LIN {X 0,Y 451.988,Z 1144.61,A -85,B 0,C 180,E1 8008.079,E2 8008.079} C_VEL
LIN {X 0,Y 452.125,Z 1144.56,A -85,B 0,C 180,E1 8011.918,E2 8011.918} C_VEL
LIN {X 0,Y 452.129,Z 1140.162,A -85,B 0,C 180,E1 8016.73,E2 8016.73} C_VEL
LIN {X 0,Y 452.581,Z 1130.609,A -85,B 0,C 180,E1 8021.579,E2 8021.579} C_VEL
LIN {X 0,Y 453.788,Z 1115.439,A -85,B 0,C 180,E1 8026.475,E2 8026.475} C_VEL
LIN {X 0,Y 456.141,Z 1093.617,A -85,B 0,C 180,E1 8031.415,E2 8031.415} C_VEL
LIN {X 0,Y 459.662,Z 1069.189,A -85,B 0,C 180,E1 8035.615,E2 8035.615} C_VEL
LIN {X 0,Y 464.182,Z 1039.886,A -85,B 0,C 180,E1 8039.437,E2 8039.437} C_VEL
LIN {X 0,Y 469.206,Z 1006.632,A -85,B 0,C 180,E1 8042.676,E2 8042.676} C_VEL
LIN {X 0,Y 474.074,Z 970.809,A -85,B 0,C 180,E1 8045.198,E2 8045.198} C_VEL
LIN {X 0,Y 477.956,Z 934.22,A -85,B 0,C 180,E1 8046.955,E2 8046.955} C_VEL
LIN {X 0,Y 479.9,Z 896.268,A -85,B 0,C 180,E1 8048.123,E2 8048.123} C_VEL
LIN {X 0,Y 466.56,Z 870.962,A -85,B 0,C 180,E1 8050.13,E2 8050.13} C_VEL
LIN {X 0,Y 451.099,Z 845.002,A -85,B 0,C 180,E1 8052.516,E2 8052.516} C_VEL
LIN {X 0,Y 450.928,Z 843.44,A -85,B 0,C 180,E1 8052.597,E2 8052.597} C_VEL
LIN {X 0,Y 450.881,Z 843.44,A -85,B 0,C 180,E1 8057.815,E2 8057.815} C_VEL
LIN {X 0,Y 450.866,Z 843.44,A -85,B 0,C 180,E1 8063.704,E2 8063.704} C_VEL
LIN {X 0,Y 450.956,Z 843.44,A -85,B 0,C 180,E1 8069.764,E2 8069.764} C_VEL
LIN {X 0,Y 451.178,Z 843.44,A -85,B 0,C 180,E1 8076.256,E2 8076.256} C_VEL
LIN {X 0,Y 451.436,Z 843.44,A -85,B 0,C 180,E1 8082.434,E2 8082.434} C_VEL
LIN {X 0,Y 451.536,Z 843.44,A -85,B 0,C 180,E1 8088.395,E2 8088.395} C_VEL
LIN {X 0,Y 451.688,Z 843.44,A -85,B 0,C 180,E1 8094.23,E2 8094.23} C_VEL
LIN {X 0,Y 451.961,Z 843.44,A -85,B 0,C 180,E1 8100.001,E2 8100.001} C_VEL
LIN {X 0,Y 451.757,Z 843.44,A -85,B 0,C 180,E1 8105.771,E2 8105.771} C_VEL
LIN {X 0,Y 451.487,Z 843.44,A -85,B 0,C 180,E1 8111.608,E2 8111.608} C_VEL
LIN {X 0,Y 451.312,Z 843.44,A -85,B 0,C 180,E1 8117.573,E2 8117.573} C_VEL
LIN {X 0,Y 451.178,Z 843.44,A -85,B 0,C 180,E1 8123.746,E2 8123.746} C_VEL
LIN {X 0,Y 450.964,Z 843.44,A -85,B 0,C 180,E1 8130.237,E2 8130.237} C_VEL
LIN {X 0,Y 450.904,Z 843.44,A -85,B 0,C 180,E1 8137.184,E2 8137.184} C_VEL
LIN {X 0,Y 450.924,Z 843.461,A -85,B 0,C 180,E1 8142.761,E2 8142.761} C_VEL
LIN {X 0,Y 453.363,Z 849.095,A -85,B 0,C 180,E1 8143.194,E2 8143.194} C_VEL
LIN {X 0,Y 471.573,Z 882.621,A -85,B 0,C 180,E1 8146.001,E2 8146.001} C_VEL
LIN {X 0,Y 482.503,Z 904.594,A -85,B 0,C 180,E1 8147.631,E2 8147.631} C_VEL
LIN {X 0,Y 479.418,Z 946.122,A -85,B 0,C 180,E1 8149.008,E2 8149.008} C_VEL
LIN {X 0,Y 475.322,Z 986.504,A -85,B 0,C 180,E1 8151.076,E2 8151.076} C_VEL
LIN {X 0,Y 473.142,Z 1005.835,A -85,B 0,C 180,E1 8152.369,E2 8152.369} C_VEL
LIN {X 0,Y 469.772,Z 1017.141,A -85,B 0,C 180,E1 8153.065,E2 8153.065} C_VEL
LIN {X 0,Y 462.499,Z 1033.593,A -85,B 0,C 180,E1 8154.101,E2 8154.101} C_VEL
LIN {X 0,Y 462.157,Z 1035.336,A -85,B 0,C 180,E1 8154.26,E2 8154.26} C_VEL
LIN {X 0,Y 456.735,Z 1071.206,A -85,B 0,C 180,E1 8158.107,E2 8158.107} C_VEL
LIN {X 0,Y 452.139,Z 1101.204,A -85,B 0,C 180,E1 8162.362,E2 8162.362} C_VEL
LIN {X 0,Y 448.304,Z 1127.32,A -85,B 0,C 180,E1 8167.408,E2 8167.408} C_VEL
LIN {X 0,Y 445.883,Z 1147.687,A -85,B 0,C 180,E1 8172.715,E2 8172.715} C_VEL
LIN {X 0,Y 444.57,Z 1162.435,A -85,B 0,C 180,E1 8178.209,E2 8178.209} C_VEL
LIN {X 0,Y 444.245,Z 1170.703,A -85,B 0,C 180,E1 8183.15,E2 8183.15} C_VEL
LIN {X 0,Y 444.193,Z 1174.657,A -85,B 0,C 180,E1 8188.047,E2 8188.047} C_VEL
LIN {X 0,Y 444.076,Z 1174.657,A -85,B 0,C 180,E1 8191.955,E2 8191.955} C_VEL
LIN {X 0,Y 444.255,Z 1170.702,A -85,B 0,C 180,E1 8196.852,E2 8196.852} C_VEL
LIN {X 0,Y 444.584,Z 1162.431,A -85,B 0,C 180,E1 8201.792,E2 8201.792} C_VEL
LIN {X 0,Y 445.785,Z 1147.68,A -85,B 0,C 180,E1 8207.29,E2 8207.29} C_VEL
LIN {X 0,Y 448.363,Z 1126.167,A -85,B 0,C 180,E1 8212.853,E2 8212.853} C_VEL
LIN {X 0,Y 452.417,Z 1099.352,A -85,B 0,C 180,E1 8217.941,E2 8217.941} C_VEL
LIN {X 0,Y 457.214,Z 1068.161,A -85,B 0,C 180,E1 8222.266,E2 8222.266} C_VEL
LIN {X 0,Y 462.623,Z 1032.575,A -85,B 0,C 180,E1 8225.99,E2 8225.99} C_VEL
LIN {X 0,Y 467.798,Z 994.238,A -85,B 0,C 180,E1 8228.965,E2 8228.965} C_VEL
LIN {X 0,Y 472.594,Z 951.617,A -85,B 0,C 180,E1 8231.307,E2 8231.307} C_VEL
LIN {X 0,Y 476.084,Z 910.219,A -85,B 0,C 180,E1 8232.791,E2 8232.791} C_VEL
LIN {X 0,Y 475.174,Z 904.691,A -85,B 0,C 180,E1 8233.045,E2 8233.045} C_VEL
LIN {X 0,Y 451.406,Z 859.546,A -85,B 0,C 180,E1 8236.811,E2 8236.811} C_VEL
LIN {X 0,Y 442.927,Z 844.493,A -85,B 0,C 180,E1 8238.251,E2 8238.251} C_VEL
LIN {X 0,Y 442.831,Z 843.44,A -85,B 0,C 180,E1 8238.363,E2 8238.363} C_VEL
LIN {X 0,Y 443.096,Z 843.44,A -85,B 0,C 180,E1 8245.098,E2 8245.098} C_VEL
LIN {X 0,Y 443.153,Z 843.44,A -85,B 0,C 180,E1 8251.426,E2 8251.426} C_VEL
LIN {X 0,Y 443.223,Z 843.52,A -85,B 0,C 180,E1 8256.584,E2 8256.584} C_VEL
LIN {X 0,Y 452.519,Z 880.617,A -85,B 0,C 180,E1 8257.692,E2 8257.692} C_VEL
LIN {X 0,Y 452.174,Z 914.08,A -85,B 0,C 180,E1 8258.568,E2 8258.568} C_VEL
LIN {X 0,Y 451.207,Z 943.567,A -85,B 0,C 180,E1 8260.103,E2 8260.103} C_VEL
LIN {X 0,Y 449.697,Z 970.782,A -85,B 0,C 180,E1 8262.362,E2 8262.362} C_VEL
LIN {X 0,Y 448.142,Z 992.836,A -85,B 0,C 180,E1 8265.072,E2 8265.072} C_VEL
LIN {X 0,Y 446.847,Z 1010.663,A -85,B 0,C 180,E1 8268.27,E2 8268.27} C_VEL
LIN {X 0,Y 445.913,Z 1023.364,A -85,B 0,C 180,E1 8271.703,E2 8271.703} C_VEL
LIN {X 0,Y 445.486,Z 1030.999,A -85,B 0,C 180,E1 8275.125,E2 8275.125} C_VEL
LIN {X 0,Y 445.205,Z 1034.117,A -85,B 0,C 180,E1 8278.05,E2 8278.05} C_VEL
LIN {X 0,Y 445.2,Z 1033.685,A -85,B 0,C 180,E1 8281.948,E2 8281.948} C_VEL
LIN {X 0,Y 445.404,Z 1028.046,A -85,B 0,C 180,E1 8285.852,E2 8285.852} C_VEL
LIN {X 0,Y 445.976,Z 1016.627,A -85,B 0,C 180,E1 8289.771,E2 8289.771} C_VEL
LIN {X 0,Y 447.074,Z 1000.684,A -85,B 0,C 180,E1 8293.212,E2 8293.212} C_VEL
LIN {X 0,Y 448.677,Z 978.808,A -85,B 0,C 180,E1 8296.414,E2 8296.414} C_VEL
LIN {X 0,Y 450.435,Z 953.007,A -85,B 0,C 180,E1 8299.001,E2 8299.001} C_VEL
LIN {X 0,Y 452.002,Z 923.588,A -85,B 0,C 180,E1 8300.954,E2 8300.954} C_VEL
LIN {X 0,Y 452.982,Z 893.055,A -85,B 0,C 180,E1 8302.152,E2 8302.152} C_VEL
LIN {X 0,Y 452.354,Z 874.82,A -85,B 0,C 180,E1 8302.58,E2 8302.58} C_VEL
LIN {X 0,Y 443.238,Z 843.44,A -85,B 0,C 180,E1 8303.639,E2 8303.639} C_VEL
LIN {X 0,Y 443.023,Z 843.44,A -85,B 0,C 180,E1 8310.836,E2 8310.836} C_VEL
LIN {X 0,Y 443.05,Z 843.44,A -85,B 0,C 180,E1 8315.513,E2 8315.513} C_VEL
LIN {X 0,Y 442.788,Z 843.44,A -85,B 0,C 180,E1 8321.209,E2 8321.209} C_VEL
LIN {X 0,Y 442.893,Z 843.44,A -85,B 0,C 180,E1 8326.27,E2 8326.27} C_VEL
LIN {X 0,Y 445.221,Z 849.073,A -85,B 0,C 180,E1 8326.711,E2 8326.711} C_VEL
LIN {X 0,Y 471.907,Z 893.713,A -85,B 0,C 180,E1 8330.848,E2 8330.848} C_VEL
LIN {X 0,Y 474.288,Z 901.421,A -85,B 0,C 180,E1 8331.306,E2 8331.306} C_VEL
LIN {X 0,Y 471.377,Z 940.453,A -85,B 0,C 180,E1 8332.537,E2 8332.537} C_VEL
LIN {X 0,Y 467.19,Z 977.315,A -85,B 0,C 180,E1 8334.454,E2 8334.454} C_VEL
LIN {X 0,Y 461.933,Z 1013.107,A -85,B 0,C 180,E1 8337.163,E2 8337.163} C_VEL
LIN {X 0,Y 456.443,Z 1045.81,A -85,B 0,C 180,E1 8340.569,E2 8340.569} C_VEL
LIN {X 0,Y 451.786,Z 1073.62,A -85,B 0,C 180,E1 8344.435,E2 8344.435} C_VEL
LIN {X 0,Y 448.042,Z 1098.182,A -85,B 0,C 180,E1 8348.956,E2 8348.956} C_VEL
LIN {X 0,Y 445.78,Z 1117.481,A -85,B 0,C 180,E1 8353.726,E2 8353.726} C_VEL
LIN {X 0,Y 444.678,Z 1131.961,A -85,B 0,C 180,E1 8358.708,E2 8358.708} C_VEL
LIN {X 0,Y 444.27,Z 1140.28,A -85,B 0,C 180,E1 8363.148,E2 8363.148} C_VEL
LIN {X 0,Y 444.084,Z 1144.609,A -85,B 0,C 180,E1 8368.045,E2 8368.045} C_VEL
LIN {X 0,Y 444.218,Z 1144.561,A -85,B 0,C 180,E1 8371.952,E2 8371.952} C_VEL
LIN {X 0,Y 444.25,Z 1140.163,A -85,B 0,C 180,E1 8376.85,E2 8376.85} C_VEL
LIN {X 0,Y 444.735,Z 1130.611,A -85,B 0,C 180,E1 8381.786,E2 8381.786} C_VEL
LIN {X 0,Y 446.046,Z 1115.443,A -85,B 0,C 180,E1 8386.77,E2 8386.77} C_VEL
LIN {X 0,Y 448.656,Z 1094.186,A -85,B 0,C 180,E1 8391.791,E2 8391.791} C_VEL
LIN {X 0,Y 452.727,Z 1068.255,A -85,B 0,C 180,E1 8396.304,E2 8396.304} C_VEL
LIN {X 0,Y 457.411,Z 1040.17,A -85,B 0,C 180,E1 8400.004,E2 8400.004} C_VEL
LIN {X 0,Y 462.775,Z 1007.287,A -85,B 0,C 180,E1 8403.257,E2 8403.257} C_VEL
LIN {X 0,Y 467.892,Z 971.936,A -85,B 0,C 180,E1 8405.78,E2 8405.78} C_VEL
LIN {X 0,Y 471.968,Z 935.502,A -85,B 0,C 180,E1 8407.555,E2 8407.555} C_VEL
LIN {X 0,Y 473.865,Z 898.713,A -85,B 0,C 180,E1 8408.731,E2 8408.731} C_VEL
LIN {X 0,Y 458.269,Z 870.375,A -85,B 0,C 180,E1 8411.114,E2 8411.114} C_VEL
LIN {X 0,Y 443.253,Z 845.31,A -85,B 0,C 180,E1 8413.536,E2 8413.536} C_VEL
LIN {X 0,Y 443.033,Z 843.44,A -85,B 0,C 180,E1 8413.664,E2 8413.664} C_VEL
LIN {X 0,Y 442.891,Z 843.44,A -85,B 0,C 180,E1 8419.499,E2 8419.499} C_VEL
LIN {X 0,Y 442.949,Z 843.44,A -85,B 0,C 180,E1 8425.123,E2 8425.123} C_VEL
LIN {X 0,Y 443.066,Z 843.44,A -85,B 0,C 180,E1 8431.422,E2 8431.422} C_VEL
LIN {X 0,Y 443.311,Z 843.44,A -85,B 0,C 180,E1 8437.936,E2 8437.936} C_VEL
LIN {X 0,Y 443.541,Z 843.44,A -85,B 0,C 180,E1 8444.154,E2 8444.154} C_VEL
LIN {X 0,Y 443.712,Z 843.44,A -85,B 0,C 180,E1 8450.178,E2 8450.178} C_VEL
LIN {X 0,Y 443.982,Z 843.44,A -85,B 0,C 180,E1 8456.09,E2 8456.09} C_VEL
LIN {X 0,Y 444.074,Z 843.44,A -85,B 0,C 180,E1 8461.955,E2 8461.955} C_VEL
LIN {X 0,Y 443.695,Z 843.44,A -85,B 0,C 180,E1 8468.26,E2 8468.26} C_VEL
LIN {X 0,Y 443.494,Z 843.44,A -85,B 0,C 180,E1 8473.826,E2 8473.826} C_VEL
LIN {X 0,Y 443.354,Z 843.44,A -85,B 0,C 180,E1 8479.968,E2 8479.968} C_VEL
LIN {X 0,Y 443.171,Z 843.44,A -85,B 0,C 180,E1 8486.367,E2 8486.367} C_VEL
LIN {X 0,Y 442.973,Z 843.44,A -85,B 0,C 180,E1 8493.151,E2 8493.151} C_VEL
LIN {X 0,Y 442.924,Z 843.44,A -85,B 0,C 180,E1 8498.165,E2 8498.165} C_VEL
LIN {X 0,Y 442.938,Z 843.44,A -85,B 0,C 180,E1 8501.704,E2 8501.704} C_VEL
LIN {X 0,Y 445.494,Z 849.185,A -85,B 0,C 180,E1 8502.203,E2 8502.203} C_VEL
LIN {X 0,Y 464.389,Z 883.185,A -85,B 0,C 180,E1 8505.243,E2 8505.243} C_VEL
LIN {X 0,Y 476.067,Z 906.688,A -85,B 0,C 180,E1 8507.099,E2 8507.099} C_VEL
LIN {X 0,Y 472.59,Z 950.335,A -85,B 0,C 180,E1 8508.627,E2 8508.627} C_VEL
LIN {X 0,Y 468.076,Z 991.225,A -85,B 0,C 180,E1 8510.839,E2 8510.839} C_VEL
LIN {X 0,Y 463.096,Z 1028.91,A -85,B 0,C 180,E1 8513.688,E2 8513.688} C_VEL
LIN {X 0,Y 462.157,Z 1035.336,A -85,B 0,C 180,E1 8514.26,E2 8514.26} C_VEL
LIN {X 0,Y 456.562,Z 1049.344,A -85,B 0,C 180,E1 8515.391,E2 8515.391} C_VEL
LIN {X 0,Y 450.91,Z 1062.707,A -85,B 0,C 180,E1 8516.626,E2 8516.626} C_VEL
LIN {X 0,Y 445.795,Z 1094.094,A -85,B 0,C 180,E1 8520.835,E2 8520.835} C_VEL
LIN {X 0,Y 441.762,Z 1119.703,A -85,B 0,C 180,E1 8525.341,E2 8525.341} C_VEL
LIN {X 0,Y 438.766,Z 1140.703,A -85,B 0,C 180,E1 8530.34,E2 8530.34} C_VEL
LIN {X 0,Y 437.189,Z 1156.564,A -85,B 0,C 180,E1 8535.511,E2 8535.511} C_VEL
LIN {X 0,Y 436.477,Z 1167.823,A -85,B 0,C 180,E1 8540.959,E2 8540.959} C_VEL
LIN {X 0,Y 436.222,Z 1173.627,A -85,B 0,C 180,E1 8546.02,E2 8546.02} C_VEL
LIN {X 0,Y 436.249,Z 1175,A -85,B 0,C 180,E1 8550.001,E2 8550.001} C_VEL
LIN {X 0,Y 436.207,Z 1173.627,A -85,B 0,C 180,E1 8553.982,E2 8553.982} C_VEL
LIN {X 0,Y 436.48,Z 1167.824,A -85,B 0,C 180,E1 8559.041,E2 8559.041} C_VEL
LIN {X 0,Y 437.211,Z 1156.56,A -85,B 0,C 180,E1 8564.491,E2 8564.491} C_VEL
LIN {X 0,Y 438.859,Z 1140.692,A -85,B 0,C 180,E1 8569.658,E2 8569.658} C_VEL
LIN {X 0,Y 442.147,Z 1117.844,A -85,B 0,C 180,E1 8575.037,E2 8575.037} C_VEL
LIN {X 0,Y 446.588,Z 1089.293,A -85,B 0,C 180,E1 8579.894,E2 8579.894} C_VEL
LIN {X 0,Y 451.984,Z 1056.085,A -85,B 0,C 180,E1 8584.135,E2 8584.135} C_VEL
LIN {X 0,Y 457.641,Z 1019.12,A -85,B 0,C 180,E1 8587.659,E2 8587.659} C_VEL
LIN {X 0,Y 463.006,Z 979.275,A -85,B 0,C 180,E1 8590.444,E2 8590.444} C_VEL
LIN {X 0,Y 467.494,Z 936.62,A -85,B 0,C 180,E1 8592.525,E2 8592.525} C_VEL
LIN {X 0,Y 469.362,Z 908.587,A -85,B 0,C 180,E1 8593.5,E2 8593.5} C_VEL
LIN {X 0,Y 446.837,Z 864.943,A -85,B 0,C 180,E1 8597.258,E2 8597.258} C_VEL
LIN {X 0,Y 435.234,Z 845.561,A -85,B 0,C 180,E1 8599.274,E2 8599.274} C_VEL
LIN {X 0,Y 434.953,Z 843.44,A -85,B 0,C 180,E1 8599.517,E2 8599.517} C_VEL
LIN {X 0,Y 435.199,Z 843.44,A -85,B 0,C 180,E1 8606.618,E2 8606.618} C_VEL
LIN {X 0,Y 435.232,Z 843.44,A -85,B 0,C 180,E1 8613.114,E2 8613.114} C_VEL
LIN {X 0,Y 435.311,Z 843.629,A -85,B 0,C 180,E1 8616.163,E2 8616.163} C_VEL
LIN {X 0,Y 445.065,Z 882.331,A -85,B 0,C 180,E1 8617.38,E2 8617.38} C_VEL
LIN {X 0,Y 444.794,Z 914.188,A -85,B 0,C 180,E1 8618.208,E2 8618.208} C_VEL
LIN {X 0,Y 443.792,Z 944.131,A -85,B 0,C 180,E1 8619.756,E2 8619.756} C_VEL
